C01813=1150.648,329.921,-76.910,-176.647,8.812,148.784
C01814=1150.652,329.674,-76.877,-176.650,8.808,148.783
C01815=1150.656,329.426,-76.845,-176.652,8.805,148.783
C01816=1150.660,329.178,-76.812,-176.654,8.801,148.783
C01817=1150.664,328.930,-76.779,-176.657,8.797,148.783
C01818=1150.668,328.682,-76.746,-176.659,8.794,148.783
C01819=1150.672,328.434,-76.713,-176.662,8.790,148.782
C01820=1150.676,328.187,-76.681,-176.665,8.787,148.782
C01821=1150.680,327.939,-76.648,-176.667,8.783,148.782
C01822=1150.684,327.690,-76.615,-176.670,8.779,148.782
C01823=1150.688,327.443,-76.582,-176.672,8.776,148.782
C01824=1150.692,327.195,-76.549,-176.675,8.772,148.781
C01825=1150.696,326.947,-76.517,-176.677,8.769,148.781
C01826=1150.700,326.699,-76.484,-176.680,8.765,148.781
C01827=1150.704,326.451,-76.452,-176.683,8.761,148.781
C01828=1150.708,326.203,-76.419,-176.685,8.758,148.781
C01829=1150.712,325.956,-76.386,-176.687,8.755,148.780
C01830=1150.717,325.708,-76.354,-176.690,8.751,148.780
C01831=1150.721,325.461,-76.321,-176.693,8.748,148.780
C01832=1150.725,325.212,-76.289,-176.696,8.744,148.780
C01833=1150.729,324.965,-76.256,-176.698,8.740,148.780
C01834=1150.733,324.717,-76.224,-176.700,8.737,148.780
C01835=1150.737,324.469,-76.190,-176.703,8.733,148.779
C01836=1150.741,324.221,-76.159,-176.706,8.730,148.779
C01837=1150.745,323.973,-76.125,-176.708,8.727,148.779
C01838=1150.749,323.726,-76.094,-176.711,8.722,148.779
C01839=1150.754,323.477,-76.062,-176.713,8.719,148.778
C01840=1150.758,323.230,-76.028,-176.716,8.715,148.778
C01841=1150.762,322.982,-75.997,-176.718,8.712,148.778
C01842=1150.766,322.734,-75.963,-176.721,8.709,148.778
C01843=1150.770,322.486,-75.932,-176.724,8.704,148.778
C01844=1150.774,322.237,-75.899,-176.726,8.701,148.778
C01845=1150.778,321.991,-75.867,-176.729,8.698,148.777
C01846=1150.783,321.742,-75.834,-176.732,8.694,148.777
C01847=1150.786,321.494,-75.803,-176.734,8.691,148.777
C01848=1150.790,321.247,-75.769,-176.736,8.688,148.777
C01849=1150.794,320.999,-75.738,-176.739,8.683,148.777
C01850=1150.799,320.751,-75.706,-176.742,8.680,148.776
C01851=1150.803,320.503,-75.674,-176.744,8.677,148.776
C01852=1150.807,320.255,-75.641,-176.747,8.673,148.776
C01853=1150.811,320.007,-75.609,-176.750,8.670,148.776
C01854=1150.815,319.759,-75.576,-176.752,8.667,148.776
C01855=1150.819,319.511,-75.545,-176.755,8.663,148.776
C01856=1150.823,319.263,-75.513,-176.757,8.659,148.775
C01857=1150.827,319.016,-75.480,-176.759,8.656,148.775
C01858=1150.831,318.768,-75.448,-176.762,8.652,148.775
C01859=1150.836,318.520,-75.416,-176.765,8.649,148.775
C01860=1150.840,318.272,-75.384,-176.767,8.646,148.775
C01861=1150.843,318.024,-75.352,-176.770,8.642,148.775
C01862=1150.848,317.776,-75.320,-176.773,8.638,148.774
C01863=1150.852,317.528,-75.288,-176.775,8.635,148.774
C01864=1150.857,317.280,-75.256,-176.778,8.631,148.774
C01865=1150.860,317.032,-75.224,-176.781,8.628,148.774
C01866=1150.865,316.785,-75.192,-176.783,8.625,148.774
C01867=1150.869,316.536,-75.160,-176.786,8.621,148.774
C01868=1150.873,316.288,-75.128,-176.788,8.617,148.773
C01869=1150.877,316.041,-75.097,-176.790,8.614,148.773
C01870=1150.881,315.793,-75.065,-176.794,8.610,148.773
C01871=1150.885,315.544,-75.032,-176.796,8.607,148.773
C01872=1150.890,315.297,-75.001,-176.798,8.604,148.773
C01873=1150.893,315.049,-74.969,-176.801,8.600,148.773
C01874=1150.898,314.801,-74.937,-176.804,8.596,148.772
C01875=1150.902,314.553,-74.905,-176.806,8.593,148.772
C01876=1150.906,314.305,-74.873,-176.809,8.590,148.772
C01877=1150.909,314.057,-74.841,-176.812,8.586,148.772
C01878=1150.914,313.779,-74.805,-176.814,8.583,148.772
C01879=1150.919,313.503,-74.770,-176.817,8.579,148.772
C01880=1150.924,313.224,-74.735,-176.820,8.575,148.772
C01881=1150.928,312.947,-74.700,-176.823,8.571,148.771
C01882=1150.932,312.699,-74.668,-176.825,8.568,148.771
C01883=1150.936,312.452,-74.636,-176.828,8.564,148.771
C01884=1150.941,312.203,-74.604,-176.831,8.561,148.771
C01885=1150.945,311.955,-74.573,-176.833,8.557,148.771
C01886=1150.949,311.707,-74.541,-176.836,8.554,148.771
C01887=1150.953,311.460,-74.510,-176.839,8.550,148.771
C01888=1150.957,311.212,-74.478,-176.841,8.547,148.770
C01889=1150.961,310.963,-74.447,-176.844,8.544,148.770
C01890=1150.966,310.716,-74.415,-176.846,8.540,148.770
C01891=1150.970,310.467,-74.383,-176.849,8.537,148.770
C01892=1150.974,310.220,-74.352,-176.852,8.533,148.770
C01893=1150.978,309.971,-74.320,-176.854,8.530,148.770
C01894=1150.983,309.724,-74.289,-176.857,8.526,148.769
C01895=1150.987,309.475,-74.258,-176.860,8.523,148.769
C01896=1150.991,309.228,-74.226,-176.862,8.520,148.769
C01897=1150.995,308.980,-74.195,-176.864,8.516,148.769
C01898=1150.999,308.731,-74.163,-176.868,8.513,148.769
C01899=1151.003,308.484,-74.132,-176.870,8.509,148.769
C01900=1151.007,308.235,-74.100,-176.872,8.506,148.769
C01901=1151.011,307.988,-74.069,-176.875,8.503,148.768
C01902=1151.015,307.739,-74.038,-176.878,8.499,148.768
C01903=1151.020,307.492,-74.006,-176.880,8.496,148.768
C01904=1151.024,307.243,-73.975,-176.883,8.493,148.768
C01905=1151.029,306.996,-73.943,-176.885,8.490,148.768
C01906=1151.033,306.747,-73.912,-176.888,8.486,148.768
C01907=1151.037,306.500,-73.881,-176.891,8.482,148.768
C01908=1151.041,306.252,-73.850,-176.893,8.479,148.768
C01909=1151.045,306.004,-73.819,-176.896,8.476,148.768
C01910=1151.049,305.756,-73.788,-176.899,8.472,148.767
C01911=1151.053,305.508,-73.757,-176.901,8.469,148.767
C01912=1151.057,305.260,-73.725,-176.904,8.466,148.767
C01913=1151.061,305.012,-73.694,-176.906,8.462,148.767
C01914=1151.066,304.764,-73.663,-176.909,8.459,148.767
C01915=1151.070,304.516,-73.631,-176.912,8.455,148.767
C01916=1151.074,304.268,-73.601,-176.914,8.452,148.767
C01917=1151.079,304.020,-73.570,-176.917,8.449,148.767
C01918=1151.083,303.772,-73.538,-176.920,8.445,148.766
C01919=1151.087,303.524,-73.507,-176.922,8.442,148.766
C01920=1151.091,303.275,-73.476,-176.925,8.439,148.766
C01921=1151.095,303.027,-73.446,-176.927,8.436,148.766
C01922=1151.099,302.780,-73.415,-176.930,8.432,148.766
C01923=1151.103,302.531,-73.383,-176.933,8.429,148.766
C01924=1151.108,302.283,-73.353,-176.935,8.426,148.766
C01925=1151.112,302.035,-73.322,-176.938,8.422,148.766
C01926=1151.117,301.787,-73.291,-176.940,8.419,148.766
C01927=1151.121,301.539,-73.261,-176.943,8.415,148.766
C01928=1151.124,301.291,-73.229,-176.946,8.412,148.765
C01929=1151.129,301.043,-73.198,-176.949,8.409,148.765
C01930=1151.134,300.795,-73.167,-176.951,8.406,148.765
C01931=1151.138,300.546,-73.136,-176.954,8.402,148.765
C01932=1151.141,300.299,-73.106,-176.957,8.399,148.765
C01933=1151.146,300.051,-73.075,-176.959,8.396,148.765
C01934=1151.150,299.802,-73.044,-176.962,8.393,148.765
C01935=1151.155,299.554,-73.013,-176.964,8.389,148.765
C01936=1151.159,299.307,-72.983,-176.967,8.385,148.765
C01937=1151.163,299.058,-72.952,-176.970,8.382,148.765
C01938=1151.167,298.810,-72.921,-176.972,8.379,148.764
C01939=1151.171,298.562,-72.891,-176.975,8.376,148.764
C01940=1151.175,298.314,-72.860,-176.977,8.373,148.764
C01941=1151.180,298.066,-72.829,-176.980,8.369,148.764
C01942=1151.184,297.818,-72.799,-176.983,8.366,148.764
C01943=1151.188,297.570,-72.768,-176.985,8.363,148.764
C01944=1151.192,297.321,-72.737,-176.988,8.360,148.764
C01945=1151.196,297.074,-72.707,-176.990,8.356,148.764
C01946=1151.201,296.826,-72.676,-176.993,8.352,148.764
C01947=1151.205,296.578,-72.645,-176.996,8.349,148.764
C01948=1151.209,296.330,-72.615,-176.999,8.346,148.764
C01949=1151.213,296.082,-72.584,-177.001,8.343,148.763
C01950=1151.217,295.834,-72.554,-177.004,8.340,148.763
C01951=1151.222,295.585,-72.524,-177.006,8.337,148.763
C01952=1151.225,295.337,-72.493,-177.009,8.333,148.763
C01953=1151.230,295.089,-72.463,-177.012,8.330,148.763
C01954=1151.234,294.841,-72.432,-177.014,8.327,148.763
C01955=1151.238,294.593,-72.402,-177.017,8.324,148.763
C01956=1151.243,294.344,-72.371,-177.019,8.321,148.763
C01957=1151.246,294.097,-72.341,-177.022,8.316,148.763
C01958=1151.251,293.849,-72.310,-177.025,8.314,148.763
C01959=1151.255,293.601,-72.280,-177.027,8.310,148.763
C01960=1151.260,293.352,-72.250,-177.030,8.307,148.763
C01961=1151.263,293.104,-72.220,-177.033,8.304,148.762
C01962=1151.268,292.856,-72.189,-177.035,8.301,148.763
C01963=1151.272,292.608,-72.159,-177.038,8.297,148.762
C01964=1151.277,292.360,-72.129,-177.041,8.294,148.762
C01965=1151.280,292.112,-72.098,-177.043,8.291,148.762
C01966=1151.285,291.863,-72.068,-177.046,8.288,148.762
C01967=1151.289,291.615,-72.038,-177.048,8.285,148.762
C01968=1151.293,291.367,-72.008,-177.051,8.282,148.762
C01969=1151.297,291.119,-71.978,-177.054,8.278,148.762
C01970=1151.301,290.871,-71.947,-177.057,8.275,148.762
C01971=1151.306,290.623,-71.917,-177.060,8.272,148.762
C01972=1151.310,290.375,-71.887,-177.062,8.268,148.762
C01973=1151.314,290.126,-71.857,-177.065,8.265,148.762
C01974=1151.318,289.878,-71.827,-177.067,8.262,148.762
C01975=1151.322,289.630,-71.797,-177.070,8.259,148.762
C01976=1151.327,289.382,-71.766,-177.073,8.255,148.761
C01977=1151.331,289.134,-71.737,-177.075,8.252,148.762
C01978=1151.335,288.886,-71.707,-177.078,8.249,148.762
C01979=1151.340,288.637,-71.677,-177.081,8.246,148.761
C01980=1151.344,288.390,-71.647,-177.083,8.243,148.761
C01981=1151.348,288.142,-71.617,-177.086,8.240,148.761
C01982=1151.352,287.866,-71.583,-177.089,8.236,148.761
C01983=1151.358,287.590,-71.550,-177.092,8.233,148.761
C01984=1151.363,287.316,-71.517,-177.095,8.229,148.761
C01985=1151.367,287.040,-71.484,-177.098,8.225,148.761
C01986=1151.371,286.793,-71.454,-177.101,8.222,148.761
C01987=1151.376,286.544,-71.425,-177.103,8.219,148.761
C01988=1151.380,286.296,-71.395,-177.106,8.216,148.761
C01989=1151.384,286.047,-71.364,-177.108,8.213,148.761
C01990=1151.388,285.799,-71.335,-177.111,8.210,148.761
C01991=1151.392,285.551,-71.305,-177.114,8.207,148.761
C01992=1151.397,285.302,-71.275,-177.117,8.203,148.761
C01993=1151.401,285.055,-71.245,-177.119,8.200,148.761
C01994=1151.405,284.806,-71.216,-177.122,8.197,148.761
C01995=1151.409,284.558,-71.186,-177.124,8.194,148.761
C01996=1151.413,284.310,-71.157,-177.127,8.191,148.761
C01997=1151.418,284.062,-71.127,-177.130,8.187,148.761
C01998=1151.422,283.814,-71.096,-177.132,8.184,148.761
C01999=1151.426,283.565,-71.067,-177.135,8.181,148.761
C02000=1151.431,283.318,-71.038,-177.137,8.178,148.760
C02001=1151.435,283.070,-71.008,-177.141,8.174,148.760
C02002=1151.440,282.821,-70.979,-177.144,8.172,148.760
C02003=1151.444,282.573,-70.950,-177.146,8.168,148.760
C02004=1151.449,282.324,-70.919,-177.149,8.165,148.760
C02005=1151.453,282.076,-70.890,-177.151,8.162,148.760
C02006=1151.457,281.829,-70.860,-177.154,8.159,148.760
C02007=1151.461,281.580,-70.830,-177.156,8.156,148.760
C02008=1151.465,281.332,-70.801,-177.159,8.153,148.760
C02009=1151.469,281.084,-70.771,-177.162,8.150,148.760
C02010=1151.473,280.835,-70.742,-177.164,8.147,148.760
C02011=1151.478,280.587,-70.713,-177.168,8.143,148.760
C02012=1151.482,280.339,-70.683,-177.170,8.140,148.760
C02013=1151.486,280.091,-70.654,-177.173,8.137,148.760
C02014=1151.491,279.843,-70.625,-177.176,8.134,148.760
C02015=1151.495,279.594,-70.596,-177.178,8.131,148.760
C02016=1151.499,279.346,-70.566,-177.181,8.128,148.760
C02017=1151.504,279.098,-70.537,-177.183,8.125,148.760
C02018=1151.508,278.849,-70.507,-177.186,8.122,148.760
C02019=1151.512,278.601,-70.478,-177.188,8.119,148.760
C02020=1151.516,278.353,-70.449,-177.191,8.116,148.760
C02021=1151.520,278.105,-70.419,-177.194,8.112,148.760
C02022=1151.524,277.856,-70.390,-177.196,8.110,148.760
C02023=1151.529,277.609,-70.361,-177.200,8.106,148.760
C02024=1151.534,277.360,-70.332,-177.202,8.103,148.760
C02025=1151.538,277.112,-70.302,-177.205,8.100,148.760
C02026=1151.542,276.863,-70.273,-177.208,8.097,148.760
C02027=1151.546,276.615,-70.243,-177.210,8.094,148.760
C02028=1151.550,276.367,-70.214,-177.213,8.091,148.760
C02029=1151.555,276.119,-70.186,-177.215,8.087,148.760
C02030=1151.559,275.871,-70.157,-177.218,8.085,148.760
C02031=1151.563,275.622,-70.127,-177.221,8.082,148.760
C02032=1151.568,275.373,-70.099,-177.223,8.078,148.760
C02033=1151.572,275.125,-70.069,-177.226,8.075,148.760
C02034=1151.577,274.878,-70.040,-177.229,8.072,148.760
C02035=1151.581,274.629,-70.011,-177.232,8.069,148.760
C02036=1151.585,274.381,-69.982,-177.234,8.066,148.760
C02037=1151.589,274.133,-69.953,-177.237,8.063,148.760
C02038=1151.593,273.884,-69.924,-177.239,8.060,148.760
C02039=1151.598,273.636,-69.895,-177.243,8.057,148.760
C02040=1151.602,273.388,-69.866,-177.246,8.054,148.760
C02041=1151.606,273.139,-69.838,-177.248,8.050,148.760
C02042=1151.610,272.891,-69.808,-177.251,8.047,148.760
C02043=1151.615,272.643,-69.780,-177.253,8.044,148.760
C02044=1151.619,272.395,-69.750,-177.256,8.042,148.760
C02045=1151.623,272.146,-69.722,-177.259,8.038,148.760
C02046=1151.628,271.898,-69.693,-177.261,8.035,148.760
C02047=1151.632,271.649,-69.664,-177.264,8.032,148.760
C02048=1151.637,271.401,-69.635,-177.267,8.029,148.760
C02049=1151.640,271.153,-69.607,-177.270,8.026,148.760
C02050=1151.645,270.905,-69.578,-177.272,8.023,148.760
C02051=1151.650,270.656,-69.549,-177.275,8.020,148.760
C02052=1151.653,270.408,-69.520,-177.278,8.017,148.760
C02053=1151.658,270.160,-69.492,-177.280,8.014,148.760
C02054=1151.662,269.912,-69.462,-177.283,8.011,148.760
C02055=1151.666,269.663,-69.434,-177.285,8.008,148.760
C02056=1151.671,269.415,-69.406,-177.288,8.005,148.760
C02057=1151.675,269.167,-69.376,-177.291,8.002,148.760
C02058=1151.679,268.918,-69.348,-177.294,7.999,148.760
C02059=1151.684,268.670,-69.320,-177.296,7.996,148.760
C02060=1151.688,268.422,-69.290,-177.299,7.993,148.760
C02061=1151.692,268.173,-69.262,-177.302,7.990,148.760
C02062=1151.697,267.925,-69.234,-177.304,7.987,148.760
C02063=1151.701,267.677,-69.204,-177.307,7.984,148.760
C02064=1151.705,267.428,-69.176,-177.310,7.981,148.760
C02065=1151.710,267.180,-69.148,-177.313,7.978,148.760
C02066=1151.714,266.931,-69.120,-177.315,7.976,148.760
C02067=1151.719,266.684,-69.091,-177.318,7.972,148.760
C02068=1151.723,266.435,-69.062,-177.321,7.969,148.760
C02069=1151.727,266.186,-69.034,-177.323,7.966,148.760
C02070=1151.731,265.938,-69.006,-177.326,7.963,148.760
C02071=1151.736,265.690,-68.977,-177.329,7.960,148.760
C02072=1151.741,265.442,-68.948,-177.332,7.958,148.760
C02073=1151.744,265.193,-68.920,-177.334,7.955,148.760
C02074=1151.749,264.945,-68.891,-177.337,7.951,148.760
C02075=1151.753,264.697,-68.863,-177.339,7.948,148.760
C02076=1151.758,264.448,-68.835,-177.342,7.945,148.760
C02077=1151.762,264.200,-68.807,-177.345,7.943,148.760
C02078=1151.766,263.951,-68.779,-177.348,7.940,148.760
C02079=1151.771,263.703,-68.750,-177.351,7.937,148.761
C02080=1151.775,263.455,-68.722,-177.353,7.934,148.761
C02081=1151.780,263.206,-68.694,-177.356,7.931,148.761
C02082=1151.783,262.958,-68.665,-177.358,7.927,148.761
C02083=1151.788,262.710,-68.637,-177.361,7.925,148.761
C02084=1151.792,262.462,-68.609,-177.364,7.922,148.761
C02085=1151.797,262.213,-68.580,-177.367,7.919,148.761
C02086=1151.802,261.940,-68.549,-177.370,7.915,148.761
C02087=1151.806,261.666,-68.518,-177.373,7.912,148.761
C02088=1151.811,261.393,-68.488,-177.376,7.909,148.761
C02089=1151.816,261.119,-68.456,-177.379,7.905,148.761
C02090=1151.820,260.871,-68.429,-177.382,7.902,148.761
C02091=1151.824,260.623,-68.401,-177.385,7.899,148.761
C02092=1151.829,260.374,-68.372,-177.387,7.896,148.761
C02093=1151.833,260.126,-68.344,-177.390,7.894,148.761
C02094=1151.837,259.878,-68.316,-177.393,7.891,148.761
C02095=1151.842,259.629,-68.288,-177.396,7.888,148.761
C02096=1151.846,259.381,-68.260,-177.398,7.886,148.761
C02097=1151.851,259.133,-68.233,-177.400,7.882,148.761
C02098=1151.854,258.884,-68.205,-177.403,7.879,148.761
C02099=1151.860,258.636,-68.176,-177.406,7.876,148.761
C02100=1151.863,258.387,-68.148,-177.409,7.873,148.761
C02101=1151.868,258.139,-68.121,-177.411,7.871,148.761
C02102=1151.872,257.890,-68.093,-177.414,7.868,148.761
C02103=1151.877,257.642,-68.064,-177.417,7.865,148.762
C02104=1151.881,257.394,-68.037,-177.420,7.862,148.762
C02105=1151.885,257.145,-68.009,-177.422,7.859,148.762
C02106=1151.890,256.897,-67.981,-177.425,7.856,148.762
C02107=1151.894,256.648,-67.953,-177.428,7.853,148.762
C02108=1151.899,256.400,-67.926,-177.431,7.850,148.762
C02109=1151.903,256.152,-67.898,-177.434,7.847,148.762
C02110=1151.907,255.903,-67.870,-177.436,7.844,148.762
C02111=1151.911,255.655,-67.843,-177.439,7.841,148.762
C02112=1151.916,255.407,-67.815,-177.442,7.838,148.762
C02113=1151.921,255.157,-67.787,-177.445,7.835,148.762
C02114=1151.925,254.910,-67.759,-177.447,7.832,148.762
C02115=1151.929,254.661,-67.731,-177.450,7.830,148.762
C02116=1151.933,254.413,-67.704,-177.452,7.827,148.762
C02117=1151.938,254.165,-67.676,-177.455,7.824,148.762
C02118=1151.942,253.915,-67.649,-177.458,7.821,148.763
C02119=1151.946,253.668,-67.621,-177.461,7.818,148.763
C02120=1151.951,253.419,-67.594,-177.464,7.816,148.763
C02121=1151.955,253.170,-67.565,-177.466,7.813,148.763
C02122=1151.960,252.922,-67.538,-177.469,7.810,148.763
C02123=1151.964,252.674,-67.510,-177.472,7.807,148.763
C02124=1151.969,252.425,-67.483,-177.475,7.804,148.763
C02125=1151.973,252.177,-67.455,-177.477,7.801,148.763
C02126=1151.977,251.928,-67.428,-177.480,7.798,148.763
C02127=1151.982,251.680,-67.400,-177.483,7.795,148.763
C02128=1151.986,251.431,-67.373,-177.485,7.793,148.763
C02129=1151.990,251.183,-67.346,-177.488,7.790,148.763
C02130=1151.995,250.935,-67.318,-177.491,7.787,148.763
C02131=1151.999,250.686,-67.291,-177.494,7.784,148.763
C02132=1152.003,250.437,-67.263,-177.496,7.781,148.764
C02133=1152.008,250.189,-67.236,-177.499,7.778,148.764
C02134=1152.012,249.941,-67.209,-177.502,7.775,148.764
C02135=1152.017,249.692,-67.182,-177.505,7.772,148.764
C02136=1152.021,249.444,-67.153,-177.507,7.769,148.764
C02137=1152.026,249.195,-67.126,-177.510,7.766,148.764
C02138=1152.030,248.947,-67.099,-177.512,7.764,148.764
C02139=1152.035,248.699,-67.072,-177.515,7.761,148.764
C02140=1152.038,248.450,-67.045,-177.518,7.758,148.764
C02141=1152.042,248.201,-67.018,-177.521,7.756,148.764
C02142=1152.047,247.953,-66.991,-177.524,7.753,148.764
C02143=1152.052,247.704,-66.964,-177.526,7.750,148.764
C02144=1152.056,247.457,-66.936,-177.529,7.747,148.764
C02145=1152.060,247.207,-66.908,-177.532,7.744,148.764
C02146=1152.065,246.959,-66.881,-177.535,7.741,148.765
C02147=1152.070,246.710,-66.854,-177.537,7.739,148.765
C02148=1152.074,246.462,-66.827,-177.540,7.736,148.765
C02149=1152.078,246.214,-66.801,-177.543,7.733,148.765
C02150=1152.083,245.965,-66.774,-177.546,7.730,148.765
C02151=1152.087,245.717,-66.745,-177.548,7.727,148.765
C02152=1152.091,245.468,-66.718,-177.551,7.724,148.765
C02153=1152.096,245.220,-66.691,-177.554,7.721,148.765
C02154=1152.100,244.971,-66.665,-177.557,7.719,148.765
C02155=1152.104,244.723,-66.638,-177.559,7.716,148.765
C02156=1152.109,244.474,-66.611,-177.562,7.714,148.766
C02157=1152.113,244.225,-66.583,-177.565,7.711,148.766
C02158=1152.118,243.977,-66.556,-177.567,7.708,148.766
C02159=1152.122,243.729,-66.530,-177.570,7.705,148.766
C02160=1152.126,243.480,-66.503,-177.573,7.702,148.766
C02161=1152.131,243.232,-66.476,-177.576,7.699,148.766
C02162=1152.136,242.983,-66.449,-177.578,7.697,148.766
C02163=1152.140,242.735,-66.422,-177.581,7.694,148.766
C02164=1152.144,242.486,-66.395,-177.584,7.691,148.766
C02165=1152.149,242.238,-66.368,-177.587,7.688,148.766
C02166=1152.153,241.989,-66.342,-177.589,7.685,148.767
C02167=1152.157,241.740,-66.315,-177.592,7.682,148.767
C02168=1152.162,241.491,-66.288,-177.594,7.680,148.767
C02169=1152.166,241.243,-66.261,-177.598,7.678,148.767
C02170=1152.170,240.995,-66.234,-177.600,7.675,148.767
C02171=1152.175,240.746,-66.207,-177.603,7.672,148.767
C02172=1152.179,240.498,-66.181,-177.606,7.669,148.767
C02173=1152.184,240.249,-66.154,-177.609,7.666,148.767
C02174=1152.189,240.000,-66.127,-177.612,7.663,148.767
C02175=1152.193,239.752,-66.101,-177.614,7.661,148.767
C02176=1152.197,239.504,-66.074,-177.617,7.658,148.768
C02177=1152.201,239.256,-66.047,-177.620,7.655,148.768
C02178=1152.206,239.006,-66.021,-177.623,7.652,148.768
C02179=1152.211,238.758,-65.994,-177.625,7.650,148.768
C02180=1152.215,238.510,-65.967,-177.628,7.647,148.768
C02181=1152.220,238.261,-65.941,-177.630,7.644,148.768
C02182=1152.224,238.013,-65.915,-177.633,7.642,148.768
C02183=1152.228,237.764,-65.888,-177.636,7.639,148.769
C02184=1152.232,237.515,-65.862,-177.639,7.636,148.769
C02185=1152.237,237.267,-65.835,-177.642,7.633,148.769
C02186=1152.241,237.019,-65.808,-177.644,7.631,148.769
C02187=1152.246,236.769,-65.782,-177.647,7.628,148.769
C02188=1152.250,236.521,-65.756,-177.650,7.625,148.769
C02189=1152.255,236.273,-65.728,-177.653,7.623,148.769
C02190=1152.260,236.001,-65.700,-177.656,7.620,148.769
C02191=1152.264,235.729,-65.671,-177.659,7.617,148.769
C02192=1152.270,235.457,-65.642,-177.661,7.614,148.770
C02193=1152.274,235.186,-65.614,-177.665,7.611,148.770
C02194=1152.279,234.937,-65.587,-177.667,7.608,148.770
C02195=1152.283,234.688,-65.561,-177.670,7.605,148.770
C02196=1152.288,234.440,-65.534,-177.673,7.602,148.770
C02197=1152.292,234.191,-65.508,-177.676,7.599,148.770
C02198=1152.296,233.943,-65.482,-177.678,7.598,148.770
C02199=1152.301,233.694,-65.455,-177.681,7.595,148.771
C02200=1152.305,233.445,-65.429,-177.684,7.592,148.771
C02201=1152.310,233.197,-65.402,-177.687,7.589,148.771
C02202=1152.314,232.948,-65.377,-177.689,7.586,148.771
C02203=1152.318,232.700,-65.351,-177.692,7.584,148.771
C02204=1152.323,232.451,-65.324,-177.695,7.581,148.771
C02205=1152.327,232.203,-65.298,-177.698,7.578,148.771
C02206=1152.332,231.954,-65.272,-177.701,7.575,148.771
C02207=1152.336,231.705,-65.246,-177.703,7.573,148.771
C02208=1152.340,231.457,-65.219,-177.706,7.571,148.772
C02209=1152.345,231.209,-65.194,-177.709,7.568,148.772
C02210=1152.350,230.960,-65.167,-177.712,7.565,148.772
C02211=1152.354,230.711,-65.141,-177.714,7.562,148.772
C02212=1152.358,230.463,-65.115,-177.717,7.560,148.772
C02213=1152.363,230.214,-65.089,-177.720,7.557,148.772
C02214=1152.368,229.965,-65.063,-177.723,7.554,148.773
C02215=1152.372,229.717,-65.037,-177.725,7.551,148.773
C02216=1152.376,229.468,-65.011,-177.728,7.549,148.773
C02217=1152.381,229.219,-64.985,-177.731,7.547,148.773
C02218=1152.385,228.971,-64.959,-177.734,7.544,148.773
C02219=1152.389,228.722,-64.933,-177.736,7.541,148.773
C02220=1152.394,228.474,-64.907,-177.739,7.539,148.773
C02221=1152.399,228.225,-64.881,-177.742,7.536,148.774
C02222=1152.403,227.976,-64.855,-177.745,7.533,148.774
C02223=1152.408,227.727,-64.829,-177.747,7.530,148.774
C02224=1152.412,227.479,-64.804,-177.750,7.528,148.774
C02225=1152.417,227.231,-64.778,-177.753,7.526,148.774
C02226=1152.421,226.982,-64.751,-177.756,7.523,148.774
C02227=1152.426,226.733,-64.726,-177.758,7.520,148.774
C02228=1152.430,226.484,-64.700,-177.761,7.518,148.774
C02229=1152.435,226.236,-64.674,-177.764,7.515,148.775
C02230=1152.439,225.988,-64.649,-177.767,7.512,148.775
C02231=1152.443,225.739,-64.623,-177.769,7.510,148.775
C02232=1152.447,225.490,-64.597,-177.772,7.507,148.775
C02233=1152.453,225.242,-64.571,-177.775,7.504,148.775
C02234=1152.457,224.993,-64.545,-177.778,7.502,148.775
C02235=1152.461,224.744,-64.520,-177.780,7.499,148.776
C02236=1152.466,224.496,-64.494,-177.783,7.497,148.776
C02237=1152.470,224.247,-64.469,-177.786,7.494,148.776
C02238=1152.475,223.998,-64.443,-177.789,7.491,148.776
C02239=1152.479,223.750,-64.417,-177.791,7.489,148.776
C02240=1152.484,223.501,-64.392,-177.794,7.486,148.776
C02241=1152.488,223.253,-64.366,-177.797,7.483,148.777
C02242=1152.492,223.004,-64.340,-177.799,7.481,148.777
C02243=1152.497,222.755,-64.315,-177.802,7.479,148.777
C02244=1152.501,222.506,-64.290,-177.805,7.476,148.777
C02245=1152.506,222.258,-64.264,-177.807,7.474,148.777
C02246=1152.510,222.009,-64.239,-177.811,7.471,148.778
C02247=1152.515,221.760,-64.213,-177.813,7.468,148.778
C02248=1152.520,221.512,-64.187,-177.816,7.465,148.778
C02249=1152.524,221.264,-64.162,-177.818,7.463,148.778
C02250=1152.528,221.014,-64.137,-177.822,7.460,148.778
C02251=1152.533,220.766,-64.111,-177.824,7.458,148.778
C02252=1152.537,220.517,-64.086,-177.827,7.455,148.778
C02253=1152.542,220.268,-64.060,-177.830,7.453,148.779
C02254=1152.547,220.020,-64.035,-177.833,7.450,148.779
C02255=1152.551,219.771,-64.009,-177.835,7.448,148.779
C02256=1152.556,219.523,-63.984,-177.838,7.445,148.779
C02257=1152.560,219.274,-63.958,-177.841,7.442,148.779
C02258=1152.564,219.025,-63.933,-177.843,7.440,148.779
C02259=1152.569,218.776,-63.908,-177.846,7.438,148.780
C02260=1152.574,218.528,-63.882,-177.849,7.435,148.780
C02261=1152.578,218.279,-63.858,-177.851,7.433,148.780
C02262=1152.582,218.030,-63.832,-177.855,7.430,148.780
C02263=1152.587,217.782,-63.807,-177.857,7.427,148.780
C02264=1152.592,217.533,-63.782,-177.860,7.425,148.780
C02265=1152.596,217.284,-63.756,-177.863,7.422,148.781
C02266=1152.601,217.035,-63.731,-177.866,7.420,148.781
C02267=1152.604,216.787,-63.706,-177.868,7.417,148.781
C02268=1152.609,216.539,-63.681,-177.871,7.415,148.781
C02269=1152.614,216.289,-63.656,-177.874,7.412,148.781
C02270=1152.619,216.041,-63.630,-177.877,7.410,148.782
C02271=1152.623,215.792,-63.605,-177.879,7.407,148.782
C02272=1152.627,215.544,-63.581,-177.882,7.404,148.782
C02273=1152.632,215.295,-63.556,-177.885,7.403,148.782
C02274=1152.637,215.047,-63.530,-177.888,7.400,148.782
C02275=1152.641,214.797,-63.505,-177.890,7.397,148.782
C02276=1152.646,214.549,-63.480,-177.893,7.395,148.783
C02277=1152.650,214.300,-63.455,-177.896,7.392,148.783
C02278=1152.654,214.052,-63.430,-177.899,7.390,148.783
C02279=1152.659,213.802,-63.405,-177.901,7.387,148.783
C02280=1152.663,213.555,-63.380,-177.904,7.384,148.783
C02281=1152.668,213.305,-63.355,-177.907,7.383,148.784
C02282=1152.673,213.056,-63.330,-177.910,7.380,148.784
C02283=1152.677,212.808,-63.305,-177.912,7.377,148.784
C02284=1152.681,212.559,-63.281,-177.915,7.375,148.784
C02285=1152.686,212.310,-63.256,-177.918,7.372,148.784
C02286=1152.691,212.062,-63.230,-177.921,7.370,148.785
C02287=1152.695,211.813,-63.206,-177.923,7.367,148.785
C02288=1152.700,211.564,-63.181,-177.926,7.364,148.785
C02289=1152.704,211.316,-63.156,-177.929,7.363,148.785
C02290=1152.708,211.067,-63.131,-177.932,7.360,148.785
C02291=1152.713,210.818,-63.107,-177.935,7.357,148.786
C02292=1152.717,210.569,-63.081,-177.937,7.355,148.786
C02293=1152.722,210.321,-63.057,-177.940,7.352,148.786
C02294=1152.727,210.050,-63.030,-177.943,7.350,148.786
C02295=1152.732,209.780,-63.003,-177.946,7.347,148.786
C02296=1152.737,209.509,-62.976,-177.949,7.345,148.787
C02297=1152.741,209.239,-62.949,-177.952,7.342,148.787
C02298=1152.747,208.990,-62.924,-177.955,7.339,148.787
C02299=1152.750,208.741,-62.900,-177.957,7.337,148.787
C02300=1152.755,208.492,-62.875,-177.960,7.335,148.787
C02301=1152.761,208.243,-62.851,-177.963,7.332,148.788
C02302=1152.764,207.994,-62.826,-177.966,7.330,148.788
C02303=1152.769,207.746,-62.801,-177.968,7.327,148.788
C02304=1152.774,207.498,-62.777,-177.972,7.325,148.788
C02305=1152.778,207.248,-62.752,-177.974,7.322,148.788
C02306=1152.783,207.000,-62.728,-177.977,7.320,148.789
C02307=1152.788,206.751,-62.703,-177.979,7.318,148.789
C02308=1152.791,206.502,-62.679,-177.982,7.315,148.789
C02309=1152.797,206.253,-62.654,-177.985,7.313,148.789
C02310=1152.801,206.005,-62.630,-177.988,7.310,148.789
C02311=1152.806,205.755,-62.605,-177.991,7.308,148.790
C02312=1152.810,205.507,-62.581,-177.993,7.306,148.790
C02313=1152.815,205.258,-62.556,-177.996,7.303,148.790
C02314=1152.819,205.009,-62.532,-177.999,7.301,148.790
C02315=1152.823,204.761,-62.508,-178.002,7.298,148.791
C02316=1152.828,204.512,-62.483,-178.004,7.296,148.791
C02317=1152.833,204.264,-62.459,-178.007,7.294,148.791
C02318=1152.837,204.014,-62.434,-178.010,7.291,148.791
C02319=1152.842,203.766,-62.410,-178.013,7.289,148.792
C02320=1152.846,203.517,-62.386,-178.016,7.286,148.792
C02321=1152.851,203.269,-62.361,-178.018,7.284,148.792
C02322=1152.855,203.020,-62.337,-178.021,7.281,148.792
C02323=1152.860,202.770,-62.313,-178.024,7.280,148.792
C02324=1152.865,202.522,-62.288,-178.027,7.277,148.793
C02325=1152.869,202.273,-62.264,-178.029,7.275,148.793
C02326=1152.874,202.024,-62.239,-178.032,7.272,148.793
C02327=1152.878,201.776,-62.215,-178.034,7.270,148.793
C02328=1152.883,201.527,-62.191,-178.037,7.267,148.794
C02329=1152.887,201.278,-62.168,-178.040,7.265,148.794
C02330=1152.892,201.029,-62.143,-178.043,7.263,148.794
C02331=1152.896,200.780,-62.119,-178.046,7.260,148.794
C02332=1152.901,200.532,-62.095,-178.048,7.258,148.794
C02333=1152.906,200.283,-62.070,-178.051,7.255,148.795
C02334=1152.910,200.034,-62.047,-178.054,7.253,148.795
C02335=1152.914,199.785,-62.022,-178.057,7.251,148.795
C02336=1152.919,199.537,-61.998,-178.059,7.249,148.795
C02337=1152.924,199.287,-61.974,-178.063,7.246,148.796
C02338=1152.928,199.039,-61.950,-178.065,7.244,148.796
C02339=1152.933,198.790,-61.926,-178.068,7.241,148.796
C02340=1152.938,198.541,-61.903,-178.070,7.239,148.796
C02341=1152.942,198.292,-61.878,-178.074,7.237,148.797
C02342=1152.946,198.044,-61.854,-178.076,7.235,148.797
C02343=1152.951,197.794,-61.830,-178.079,7.232,148.797
C02344=1152.956,197.546,-61.806,-178.081,7.230,148.797
C02345=1152.960,197.298,-61.782,-178.085,7.227,148.797
C02346=1152.965,197.049,-61.759,-178.087,7.225,148.798
C02347=1152.970,196.800,-61.734,-178.090,7.223,148.798
C02348=1152.974,196.550,-61.710,-178.092,7.221,148.798
C02349=1152.978,196.302,-61.686,-178.096,7.218,148.798
C02350=1152.983,196.053,-61.663,-178.098,7.216,148.799
C02351=1152.987,195.804,-61.639,-178.101,7.213,148.799
C02352=1152.992,195.555,-61.615,-178.104,7.212,148.799
C02353=1152.996,195.307,-61.591,-178.106,7.209,148.799
C02354=1153.002,195.058,-61.567,-178.109,7.207,148.800
C02355=1153.006,194.809,-61.543,-178.112,7.204,148.800
C02356=1153.011,194.560,-61.520,-178.115,7.202,148.800
C02357=1153.015,194.312,-61.496,-178.117,7.199,148.800
C02358=1153.020,194.063,-61.473,-178.120,7.198,148.801
C02359=1153.024,193.814,-61.448,-178.123,7.195,148.801
C02360=1153.029,193.564,-61.425,-178.126,7.193,148.801
C02361=1153.033,193.315,-61.401,-178.129,7.190,148.801
C02362=1153.038,193.067,-61.377,-178.131,7.188,148.802
C02363=1153.042,192.818,-61.354,-178.134,7.186,148.802
C02364=1153.047,192.570,-61.330,-178.137,7.184,148.802
C02365=1153.051,192.321,-61.307,-178.140,7.181,148.802
C02366=1153.056,192.072,-61.283,-178.143,7.179,148.803
C02367=1153.061,191.823,-61.259,-178.145,7.177,148.803
C02368=1153.065,191.574,-61.236,-178.148,7.175,148.803
C02369=1153.070,191.325,-61.212,-178.150,7.173,148.803
C02370=1153.074,191.077,-61.188,-178.153,7.170,148.804
C02371=1153.079,190.828,-61.165,-178.156,7.168,148.804
C02372=1153.084,190.579,-61.142,-178.159,7.165,148.804
C02373=1153.088,190.330,-61.118,-178.162,7.164,148.804
C02374=1153.093,190.081,-61.094,-178.164,7.161,148.805
C02375=1153.098,189.832,-61.071,-178.167,7.159,148.805
C02376=1153.102,189.583,-61.047,-178.170,7.156,148.805
C02377=1153.107,189.334,-61.024,-178.173,7.154,148.805
C02378=1153.112,189.085,-61.001,-178.175,7.152,148.806
C02379=1153.116,188.837,-60.977,-178.178,7.150,148.806
C02380=1153.121,188.588,-60.953,-178.181,7.148,148.806
C02381=1153.125,188.339,-60.931,-178.184,7.145,148.807
C02382=1153.130,188.091,-60.908,-178.186,7.143,148.807
C02383=1153.135,187.841,-60.884,-178.190,7.141,148.807
C02384=1153.139,187.592,-60.861,-178.192,7.138,148.807
C02385=1153.144,187.343,-60.837,-178.194,7.137,148.808
C02386=1153.148,187.095,-60.813,-178.198,7.134,148.808
C02387=1153.153,186.846,-60.790,-178.200,7.132,148.808
C02388=1153.157,186.597,-60.767,-178.203,7.129,148.808
C02389=1153.162,186.348,-60.744,-178.206,7.128,148.809
C02390=1153.167,186.099,-60.721,-178.209,7.125,148.809
C02391=1153.171,185.850,-60.697,-178.211,7.123,148.809
C02392=1153.176,185.601,-60.674,-178.214,7.121,148.810
C02393=1153.181,185.353,-60.651,-178.217,7.118,148.810
C02394=1153.185,185.104,-60.628,-178.220,7.117,148.810
C02395=1153.190,184.855,-60.605,-178.222,7.114,148.810
C02396=1153.195,184.606,-60.581,-178.225,7.112,148.810
C02397=1153.199,184.357,-60.559,-178.228,7.110,148.811
C02398=1153.204,184.088,-60.534,-178.231,7.108,148.811
C02399=1153.209,183.818,-60.509,-178.234,7.105,148.811
C02400=1153.215,183.548,-60.483,-178.237,7.102,148.812
C02401=1153.219,183.279,-60.458,-178.240,7.100,148.812
C02402=1153.224,183.029,-60.436,-178.243,7.098,148.812
C02403=1153.229,182.780,-60.412,-178.245,7.096,148.812
C02404=1153.232,182.532,-60.390,-178.248,7.094,148.813
C02405=1153.237,182.283,-60.366,-178.251,7.092,148.813
C02406=1153.242,182.034,-60.343,-178.253,7.089,148.813
C02407=1153.246,181.786,-60.320,-178.257,7.087,148.814
C02408=1153.251,181.537,-60.297,-178.259,7.085,148.814
C02409=1153.256,181.287,-60.274,-178.262,7.083,148.814
C02410=1153.260,181.038,-60.252,-178.265,7.080,148.815
C02411=1153.265,180.789,-60.228,-178.268,7.079,148.815
C02412=1153.270,180.541,-60.205,-178.270,7.077,148.815
C02413=1153.274,180.292,-60.183,-178.273,7.074,148.815
C02414=1153.279,180.043,-60.160,-178.276,7.072,148.816
C02415=1153.283,179.794,-60.137,-178.279,7.069,148.816
C02416=1153.288,179.545,-60.114,-178.281,7.068,148.816
C02417=1153.293,179.296,-60.091,-178.284,7.066,148.817
C02418=1153.297,179.047,-60.069,-178.287,7.063,148.817
C02419=1153.302,178.798,-60.045,-178.289,7.061,148.817
C02420=1153.306,178.549,-60.023,-178.292,7.060,148.817
C02421=1153.312,178.300,-60.000,-178.295,7.057,148.818
C02422=1153.316,178.052,-59.978,-178.298,7.055,148.818
C02423=1153.320,177.803,-59.954,-178.301,7.052,148.818
C02424=1153.326,177.554,-59.932,-178.304,7.051,148.819
C02425=1153.330,177.305,-59.909,-178.306,7.049,148.819
C02426=1153.335,177.056,-59.886,-178.309,7.046,148.819
C02427=1153.339,176.807,-59.864,-178.312,7.044,148.819
C02428=1153.344,176.558,-59.841,-178.314,7.042,148.820
C02429=1153.348,176.309,-59.819,-178.317,7.040,148.820
C02430=1153.353,176.060,-59.795,-178.320,7.038,148.820
C02431=1153.358,175.811,-59.774,-178.323,7.036,148.821
C02432=1153.363,175.562,-59.750,-178.326,7.033,148.821
C02433=1153.367,175.313,-59.728,-178.328,7.031,148.821
C02434=1153.371,175.065,-59.706,-178.331,7.030,148.822
C02435=1153.376,174.815,-59.683,-178.334,7.027,148.822
C02436=1153.380,174.566,-59.660,-178.336,7.025,148.822
C02437=1153.386,174.318,-59.638,-178.339,7.023,148.822
C02438=1153.390,174.069,-59.615,-178.342,7.021,148.823
C02439=1153.395,173.819,-59.593,-178.345,7.019,148.823
C02440=1153.400,173.571,-59.570,-178.347,7.017,148.823
C02441=1153.404,173.322,-59.548,-178.351,7.014,148.824
C02442=1153.409,173.073,-59.525,-178.353,7.013,148.824
C02443=1153.413,172.824,-59.503,-178.356,7.011,148.824
C02444=1153.418,172.574,-59.481,-178.359,7.008,148.824
C02445=1153.422,172.326,-59.458,-178.361,7.006,148.825
C02446=1153.427,172.077,-59.436,-178.364,7.004,148.825
C02447=1153.432,171.828,-59.413,-178.367,7.002,148.826
C02448=1153.437,171.579,-59.391,-178.370,7.000,148.826
C02449=1153.441,171.330,-59.369,-178.372,6.998,148.826
C02450=1153.446,171.081,-59.346,-178.375,6.996,148.826
C02451=1153.451,170.832,-59.324,-178.378,6.994,148.827
C02452=1153.455,170.583,-59.302,-178.381,6.992,148.827
C02453=1153.460,170.335,-59.279,-178.383,6.990,148.827
C02454=1153.464,170.085,-59.257,-178.386,6.987,148.828
C02455=1153.469,169.837,-59.235,-178.389,6.986,148.828
C02456=1153.474,169.587,-59.213,-178.392,6.984,148.828
C02457=1153.478,169.338,-59.190,-178.395,6.981,148.829
C02458=1153.483,169.090,-59.168,-178.397,6.979,148.829
C02459=1153.487,168.840,-59.146,-178.400,6.978,148.829
C02460=1153.493,168.591,-59.124,-178.403,6.976,148.830
C02461=1153.497,168.342,-59.102,-178.406,6.973,148.830
C02462=1153.502,168.094,-59.079,-178.408,6.971,148.830
C02463=1153.506,167.845,-59.057,-178.411,6.969,148.831
C02464=1153.511,167.596,-59.036,-178.414,6.967,148.831
C02465=1153.516,167.346,-59.013,-178.417,6.965,148.831
C02466=1153.521,167.098,-58.991,-178.419,6.963,148.831
C02467=1153.525,166.848,-58.969,-178.422,6.961,148.832
C02468=1153.530,166.600,-58.948,-178.425,6.959,148.832
C02469=1153.534,166.351,-58.925,-178.428,6.957,148.832
C02470=1153.540,166.102,-58.903,-178.431,6.955,148.833
C02471=1153.544,165.853,-58.881,-178.433,6.953,148.833
C02472=1153.549,165.604,-58.859,-178.436,6.951,148.833
C02473=1153.553,165.355,-58.837,-178.439,6.949,148.834
C02474=1153.558,165.106,-58.815,-178.441,6.947,148.834
C02475=1153.562,164.857,-58.793,-178.444,6.945,148.834
C02476=1153.567,164.608,-58.771,-178.447,6.943,148.835
C02477=1153.572,164.359,-58.749,-178.450,6.941,148.835
C02478=1153.577,164.110,-58.727,-178.452,6.939,148.835
C02479=1153.581,163.861,-58.705,-178.455,6.937,148.836
C02480=1153.586,163.612,-58.683,-178.458,6.935,148.836
C02481=1153.590,163.363,-58.661,-178.461,6.933,148.836
C02482=1153.595,163.114,-58.640,-178.464,6.931,148.837
C02483=1153.600,162.865,-58.618,-178.466,6.929,148.837
C02484=1153.604,162.616,-58.596,-178.469,6.927,148.837
C02485=1153.609,162.367,-58.574,-178.472,6.925,148.838
C02486=1153.614,162.117,-58.553,-178.475,6.923,148.838
C02487=1153.619,161.869,-58.531,-178.477,6.921,148.838
C02488=1153.623,161.619,-58.509,-178.481,6.919,148.839
C02489=1153.628,161.371,-58.487,-178.483,6.917,148.839
C02490=1153.633,161.122,-58.466,-178.486,6.915,148.839
C02491=1153.637,160.873,-58.444,-178.488,6.913,148.840
C02492=1153.642,160.624,-58.422,-178.492,6.911,148.840
C02493=1153.647,160.375,-58.401,-178.494,6.909,148.840
C02494=1153.651,160.126,-58.379,-178.497,6.907,148.841
C02495=1153.656,159.877,-58.357,-178.499,6.905,148.841
C02496=1153.660,159.628,-58.335,-178.502,6.904,148.841
C02497=1153.665,159.379,-58.314,-178.505,6.901,148.842
C02498=1153.670,159.130,-58.293,-178.508,6.899,148.842
C02499=1153.675,158.880,-58.271,-178.511,6.898,148.842
C02500=1153.680,158.632,-58.249,-178.513,6.896,148.843
C02501=1153.684,158.383,-58.227,-178.517,6.893,148.843
C02502=1153.689,158.114,-58.204,-178.519,6.892,148.844
C02503=1153.695,157.845,-58.181,-178.522,6.890,148.844
C02504=1153.699,157.576,-58.158,-178.525,6.887,148.844
C02505=1153.705,157.307,-58.134,-178.528,6.886,148.845
C02506=1153.710,157.058,-58.113,-178.531,6.883,148.845
C02507=1153.714,156.808,-58.091,-178.533,6.881,148.845
C02508=1153.718,156.560,-58.070,-178.536,6.879,148.846
C02509=1153.723,156.311,-58.049,-178.539,6.877,148.846
C02510=1153.728,156.061,-58.027,-178.542,6.876,148.846
C02511=1153.732,155.813,-58.006,-178.545,6.873,148.847
C02512=1153.738,155.563,-57.985,-178.548,6.871,148.847
C02513=1153.742,155.315,-57.963,-178.550,6.870,148.847
C02514=1153.747,155.065,-57.942,-178.553,6.868,148.848
C02515=1153.751,154.816,-57.920,-178.556,6.866,148.848
C02516=1153.756,154.568,-57.899,-178.558,6.864,148.848
C02517=1153.761,154.319,-57.878,-178.561,6.862,148.849
C02518=1153.765,154.069,-57.856,-178.564,6.860,148.849
C02519=1153.771,153.820,-57.835,-178.567,6.858,148.850
C02520=1153.775,153.572,-57.814,-178.569,6.856,148.850
C02521=1153.780,153.322,-57.793,-178.572,6.855,148.850
C02522=1153.784,153.073,-57.771,-178.575,6.852,148.851
C02523=1153.789,152.824,-57.750,-178.578,6.850,148.851
C02524=1153.794,152.575,-57.729,-178.581,6.849,148.851
C02525=1153.799,152.326,-57.708,-178.583,6.847,148.852
C02526=1153.803,152.076,-57.686,-178.586,6.845,148.852
C02527=1153.808,151.828,-57.665,-178.588,6.843,148.852
C02528=1153.813,151.579,-57.644,-178.591,6.841,148.853
C02529=1153.817,151.330,-57.623,-178.594,6.839,148.853
C02530=1153.823,151.081,-57.602,-178.597,6.837,148.853
C02531=1153.826,150.831,-57.581,-178.600,6.835,148.854
C02532=1153.831,150.582,-57.559,-178.602,6.834,148.854
C02533=1153.837,150.333,-57.538,-178.605,6.832,148.855
C02534=1153.841,150.084,-57.518,-178.608,6.830,148.855
C02535=1153.846,149.836,-57.496,-178.611,6.828,148.855
C02536=1153.851,149.586,-57.475,-178.614,6.826,148.856
C02537=1153.855,149.337,-57.454,-178.616,6.824,148.856
C02538=1153.860,149.088,-57.433,-178.619,6.823,148.856
C02539=1153.865,148.839,-57.412,-178.621,6.820,148.857
C02540=1153.869,148.590,-57.391,-178.624,6.819,148.857
C02541=1153.874,148.341,-57.370,-178.627,6.817,148.857
C02542=1153.879,148.092,-57.349,-178.630,6.815,148.858
C02543=1153.884,147.843,-57.328,-178.633,6.813,148.858
C02544=1153.888,147.593,-57.307,-178.636,6.811,148.859
C02545=1153.893,147.344,-57.287,-178.638,6.809,148.859
C02546=1153.898,147.095,-57.265,-178.641,6.808,148.859
C02547=1153.902,146.847,-57.245,-178.644,6.806,148.860
C02548=1153.907,146.597,-57.224,-178.646,6.804,148.860
C02549=1153.912,146.348,-57.203,-178.649,6.802,148.860
C02550=1153.917,146.099,-57.182,-178.652,6.801,148.861
C02551=1153.922,145.850,-57.161,-178.655,6.798,148.861
C02552=1153.926,145.601,-57.140,-178.658,6.796,148.862
C02553=1153.931,145.352,-57.119,-178.660,6.795,148.862
C02554=1153.936,145.103,-57.099,-178.663,6.793,148.862
C02555=1153.940,144.853,-57.078,-178.666,6.791,148.863
C02556=1153.945,144.604,-57.057,-178.669,6.790,148.863
C02557=1153.950,144.355,-57.036,-178.671,6.788,148.864
C02558=1153.954,144.106,-57.016,-178.674,6.786,148.864
C02559=1153.960,143.857,-56.995,-178.677,6.784,148.864
C02560=1153.964,143.608,-56.975,-178.680,6.781,148.864
C02561=1153.969,143.359,-56.954,-178.682,6.780,148.865
C02562=1153.974,143.110,-56.933,-178.685,6.778,148.865
C02563=1153.978,142.861,-56.913,-178.688,6.776,148.866
C02564=1153.983,142.611,-56.892,-178.690,6.775,148.866
C02565=1153.988,142.363,-56.872,-178.693,6.773,148.866
C02566=1153.993,142.113,-56.851,-178.696,6.771,148.867
C02567=1153.997,141.864,-56.830,-178.698,6.769,148.867
C02568=1154.002,141.615,-56.810,-178.701,6.768,148.868
C02569=1154.007,141.366,-56.789,-178.704,6.766,148.868
C02570=1154.011,141.117,-56.768,-178.707,6.764,148.868
C02571=1154.017,140.868,-56.748,-178.710,6.762,148.869
C02572=1154.021,140.619,-56.727,-178.713,6.760,148.869
C02573=1154.025,140.370,-56.707,-178.715,6.758,148.869
C02574=1154.031,140.121,-56.686,-178.718,6.757,148.870
C02575=1154.035,139.872,-56.665,-178.721,6.755,148.870
C02576=1154.039,139.623,-56.645,-178.723,6.753,148.871
C02577=1154.045,139.373,-56.625,-178.726,6.751,148.871
C02578=1154.049,139.124,-56.604,-178.729,6.750,148.871
C02579=1154.054,138.875,-56.584,-178.732,6.748,148.872
C02580=1154.059,138.626,-56.563,-178.734,6.746,148.872
C02581=1154.063,138.377,-56.543,-178.737,6.745,148.873
C02582=1154.068,138.128,-56.522,-178.740,6.743,148.873
C02583=1154.073,137.878,-56.502,-178.742,6.741,148.873
C02584=1154.078,137.629,-56.482,-178.745,6.739,148.874
C02585=1154.082,137.380,-56.461,-178.748,6.738,148.874
C02586=1154.087,137.132,-56.441,-178.751,6.736,148.875
C02587=1154.093,136.882,-56.421,-178.753,6.734,148.875
C02588=1154.097,136.633,-56.401,-178.757,6.732,148.875
C02589=1154.102,136.384,-56.380,-178.759,6.730,148.876
C02590=1154.106,136.135,-56.360,-178.762,6.728,148.876
C02591=1154.112,135.885,-56.340,-178.765,6.727,148.877
C02592=1154.116,135.636,-56.319,-178.768,6.725,148.877
C02593=1154.120,135.387,-56.299,-178.771,6.723,148.877
C02594=1154.125,135.138,-56.279,-178.773,6.722,148.878
C02595=1154.130,134.890,-56.259,-178.776,6.720,148.878
C02596=1154.135,134.640,-56.238,-178.779,6.718,148.879
C02597=1154.140,134.391,-56.219,-178.781,6.717,148.879
C02598=1154.145,134.142,-56.198,-178.784,6.715,148.879
C02599=1154.149,133.892,-56.179,-178.787,6.713,148.880
C02600=1154.154,133.643,-56.158,-178.790,6.711,148.880
C02601=1154.159,133.394,-56.137,-178.792,6.710,148.881
C02602=1154.164,133.145,-56.118,-178.795,6.708,148.881
C02603=1154.169,132.896,-56.098,-178.798,6.706,148.881
C02604=1154.173,132.647,-56.078,-178.800,6.705,148.882
C02605=1154.178,132.398,-56.058,-178.803,6.703,148.882
C02606=1154.184,132.129,-56.036,-178.806,6.701,148.883
C02607=1154.188,131.860,-56.015,-178.809,6.699,148.883
C02608=1154.193,131.592,-55.993,-178.812,6.697,148.884
C02609=1154.199,131.323,-55.971,-178.815,6.696,148.884
C02610=1154.203,131.074,-55.951,-178.818,6.694,148.884
C02611=1154.208,130.825,-55.932,-178.820,6.692,148.885
C02612=1154.213,130.576,-55.911,-178.823,6.690,148.885
C02613=1154.218,130.327,-55.892,-178.826,6.689,148.886
C02614=1154.222,130.077,-55.872,-178.829,6.687,148.886
C02615=1154.227,129.828,-55.852,-178.831,6.685,148.886
C02616=1154.232,129.579,-55.832,-178.834,6.684,148.887
C02617=1154.237,129.330,-55.812,-178.837,6.682,148.887
C02618=1154.241,129.081,-55.792,-178.839,6.680,148.888
C02619=1154.246,128.831,-55.773,-178.843,6.679,148.888
C02620=1154.251,128.583,-55.753,-178.845,6.677,148.889
C02621=1154.256,128.333,-55.733,-178.848,6.675,148.889
C02622=1154.260,128.085,-55.713,-178.851,6.674,148.889
C02623=1154.265,127.835,-55.693,-178.854,6.672,148.890
C02624=1154.270,127.586,-55.674,-178.856,6.670,148.890
C02625=1154.275,127.337,-55.653,-178.859,6.668,148.891
C02626=1154.280,127.088,-55.634,-178.862,6.667,148.891
C02627=1154.285,126.839,-55.614,-178.864,6.665,148.891
C02628=1154.290,126.589,-55.595,-178.867,6.663,148.892
C02629=1154.294,126.340,-55.574,-178.870,6.662,148.892
C02630=1154.299,126.091,-55.555,-178.873,6.660,148.893
C02631=1154.304,125.842,-55.535,-178.876,6.659,148.893
C02632=1154.309,125.592,-55.516,-178.878,6.657,148.894
C02633=1154.313,125.343,-55.495,-178.881,6.655,148.894
C02634=1154.319,125.094,-55.476,-178.884,6.653,148.894
C02635=1154.323,124.845,-55.456,-178.887,6.652,148.895
C02636=1154.327,124.596,-55.437,-178.889,6.651,148.895
C02637=1154.333,124.347,-55.417,-178.891,6.649,148.896
C02638=1154.337,124.098,-55.398,-178.894,6.647,148.896
C02639=1154.342,123.848,-55.378,-178.897,6.646,148.896
C02640=1154.347,123.599,-55.359,-178.900,6.644,148.897
C02641=1154.352,123.350,-55.339,-178.902,6.642,148.897
C02642=1154.357,123.100,-55.319,-178.905,6.641,148.898
C02643=1154.361,122.852,-55.301,-178.908,6.639,148.898
C02644=1154.366,122.603,-55.280,-178.911,6.637,148.899
C02645=1154.371,122.353,-55.261,-178.914,6.636,148.899
C02646=1154.376,122.104,-55.241,-178.916,6.634,148.899
C02647=1154.381,121.855,-55.222,-178.919,6.632,148.900
C02648=1154.385,121.605,-55.203,-178.922,6.631,148.900
C02649=1154.390,121.357,-55.183,-178.925,6.629,148.901
C02650=1154.395,121.107,-55.164,-178.928,6.628,148.901
C02651=1154.400,120.858,-55.145,-178.930,6.626,148.902
C02652=1154.405,120.609,-55.125,-178.933,6.624,148.902
C02653=1154.409,120.359,-55.106,-178.935,6.623,148.902
C02654=1154.414,120.110,-55.086,-178.938,6.622,148.903
C02655=1154.419,119.861,-55.067,-178.941,6.620,148.903
C02656=1154.424,119.612,-55.048,-178.943,6.618,148.904
C02657=1154.428,119.363,-55.028,-178.946,6.616,148.904
C02658=1154.434,119.114,-55.009,-178.949,6.615,148.905
C02659=1154.438,118.864,-54.990,-178.952,6.613,148.905
C02660=1154.442,118.615,-54.970,-178.955,6.612,148.905
C02661=1154.448,118.366,-54.951,-178.958,6.610,148.906
C02662=1154.453,118.117,-54.932,-178.960,6.608,148.906
C02663=1154.458,117.868,-54.912,-178.963,6.607,148.907
C02664=1154.462,117.618,-54.894,-178.966,6.605,148.907
C02665=1154.468,117.369,-54.875,-178.968,6.604,148.907
C02666=1154.472,117.119,-54.855,-178.971,6.603,148.908
C02667=1154.477,116.871,-54.836,-178.974,6.601,148.908
C02668=1154.482,116.621,-54.817,-178.976,6.599,148.909
C02669=1154.487,116.372,-54.797,-178.979,6.598,148.909
C02670=1154.491,116.123,-54.778,-178.982,6.596,148.910
C02671=1154.497,115.874,-54.760,-178.985,6.594,148.910
C02672=1154.501,115.624,-54.741,-178.988,6.593,148.911
C02673=1154.506,115.376,-54.721,-178.991,6.591,148.911
C02674=1154.511,115.126,-54.702,-178.993,6.590,148.912
C02675=1154.515,114.877,-54.683,-178.995,6.588,148.912
C02676=1154.520,114.627,-54.664,-178.998,6.587,148.912
C02677=1154.525,114.379,-54.645,-179.001,6.585,148.913
C02678=1154.530,114.129,-54.626,-179.004,6.583,148.913
C02679=1154.535,113.880,-54.606,-179.007,6.582,148.914
C02680=1154.539,113.630,-54.588,-179.009,6.580,148.914
C02681=1154.545,113.381,-54.569,-179.012,6.579,148.915
C02682=1154.549,113.132,-54.550,-179.015,6.577,148.915
C02683=1154.554,112.883,-54.531,-179.017,6.576,148.915
C02684=1154.558,112.633,-54.512,-179.020,6.574,148.916
C02685=1154.564,112.385,-54.493,-179.023,6.573,148.916
C02686=1154.569,112.135,-54.475,-179.026,6.571,148.917
C02687=1154.573,111.886,-54.455,-179.028,6.570,148.917
C02688=1154.579,111.637,-54.436,-179.031,6.568,148.918
C02689=1154.583,111.387,-54.417,-179.034,6.566,148.918
C02690=1154.588,111.138,-54.398,-179.036,6.565,148.918
C02691=1154.593,110.889,-54.380,-179.039,6.564,148.919
C02692=1154.597,110.640,-54.361,-179.042,6.562,148.920
C02693=1154.603,110.391,-54.342,-179.045,6.561,148.920
C02694=1154.607,110.141,-54.324,-179.047,6.559,148.920
C02695=1154.612,109.892,-54.304,-179.050,6.557,148.921
C02696=1154.617,109.643,-54.286,-179.053,6.556,148.921
C02697=1154.622,109.393,-54.267,-179.055,6.555,148.922
C02698=1154.627,109.144,-54.249,-179.058,6.553,148.922
C02699=1154.632,108.895,-54.229,-179.061,6.551,148.923
C02700=1154.636,108.646,-54.211,-179.064,6.550,148.923
C02701=1154.641,108.397,-54.192,-179.067,6.548,148.924
C02702=1154.646,108.147,-54.173,-179.070,6.547,148.924
C02703=1154.651,107.898,-54.155,-179.072,6.546,148.924
C02704=1154.656,107.649,-54.136,-179.074,6.544,148.925
C02705=1154.660,107.400,-54.117,-179.077,6.542,148.925
C02706=1154.665,107.150,-54.099,-179.080,6.541,148.926
C02707=1154.671,106.901,-54.080,-179.083,6.539,148.926
C02708=1154.675,106.652,-54.061,-179.086,6.538,148.927
C02709=1154.680,106.402,-54.043,-179.088,6.537,148.927
C02710=1154.685,106.134,-54.023,-179.091,6.535,148.928
C02711=1154.690,105.866,-54.003,-179.094,6.534,148.928
C02712=1154.696,105.597,-53.983,-179.097,6.532,148.929
C02713=1154.700,105.329,-53.963,-179.100,6.530,148.929
C02714=1154.706,105.080,-53.944,-179.102,6.529,148.930
C02715=1154.710,104.830,-53.926,-179.105,6.527,148.930
C02716=1154.715,104.581,-53.907,-179.108,6.526,148.930
C02717=1154.721,104.332,-53.889,-179.111,6.524,148.931
C02718=1154.725,104.082,-53.870,-179.114,6.523,148.932
C02719=1154.730,103.833,-53.852,-179.116,6.522,148.932
C02720=1154.735,103.584,-53.834,-179.119,6.520,148.932
C02721=1154.740,103.335,-53.815,-179.121,6.518,148.933
C02722=1154.744,103.085,-53.797,-179.125,6.517,148.933
C02723=1154.749,102.836,-53.778,-179.127,6.515,148.934
C02724=1154.754,102.587,-53.760,-179.129,6.514,148.934
C02725=1154.760,102.338,-53.741,-179.132,6.513,148.935
C02726=1154.764,102.088,-53.723,-179.135,6.511,148.935
C02727=1154.769,101.839,-53.704,-179.138,6.510,148.936
C02728=1154.773,101.590,-53.686,-179.141,6.508,148.936
C02729=1154.779,101.341,-53.668,-179.143,6.507,148.937
C02730=1154.783,101.091,-53.649,-179.146,6.505,148.937
C02731=1154.788,100.842,-53.631,-179.149,6.504,148.938
C02732=1154.793,100.593,-53.613,-179.152,6.502,148.938
C02733=1154.798,100.344,-53.595,-179.154,6.502,148.938
C02734=1154.803,100.095,-53.577,-179.157,6.500,148.939
C02735=1154.808,99.844,-53.558,-179.160,6.499,148.939
C02736=1154.813,99.595,-53.540,-179.162,6.497,148.940
C02737=1154.818,99.346,-53.522,-179.165,6.495,148.940
C02738=1154.823,99.097,-53.504,-179.167,6.494,148.941
C02739=1154.827,98.848,-53.486,-179.171,6.493,148.941
C02740=1154.831,98.599,-53.467,-179.173,6.491,148.942
C02741=1154.836,98.349,-53.449,-179.176,6.490,148.942
C02742=1154.842,98.100,-53.430,-179.178,6.489,148.943
C02743=1154.847,97.851,-53.412,-179.181,6.487,148.943
C02744=1154.852,97.602,-53.394,-179.184,6.486,148.944
C02745=1154.857,97.352,-53.376,-179.187,6.484,148.944
C02746=1154.861,97.102,-53.358,-179.189,6.483,148.944
C02747=1154.866,96.853,-53.340,-179.192,6.482,148.945
C02748=1154.871,96.604,-53.322,-179.195,6.480,148.946
C02749=1154.876,96.355,-53.304,-179.198,6.478,148.946
C02750=1154.881,96.106,-53.286,-179.200,6.477,148.946
C02751=1154.886,95.857,-53.268,-179.203,6.476,148.947
C02752=1154.891,95.607,-53.250,-179.206,6.474,148.947
C02753=1154.895,95.358,-53.232,-179.208,6.473,148.948
C02754=1154.900,95.108,-53.214,-179.211,6.472,148.948
C02755=1154.905,94.859,-53.196,-179.214,6.471,148.949
C02756=1154.910,94.609,-53.179,-179.217,6.469,148.949
C02757=1154.915,94.360,-53.161,-179.219,6.467,148.950
C02758=1154.920,94.111,-53.143,-179.221,6.466,148.950
C02759=1154.925,93.862,-53.125,-179.225,6.465,148.951
C02760=1154.930,93.613,-53.107,-179.227,6.463,148.951
C02761=1154.934,93.364,-53.089,-179.230,6.462,148.952
C02762=1154.939,93.114,-53.071,-179.232,6.461,148.952
C02763=1154.944,92.865,-53.053,-179.235,6.459,148.953
C02764=1154.949,92.615,-53.035,-179.238,6.458,148.953
C02765=1154.954,92.365,-53.017,-179.240,6.457,148.954
C02766=1154.959,92.116,-52.999,-179.243,6.455,148.954
C02767=1154.964,91.867,-52.981,-179.246,6.454,148.955
C02768=1154.969,91.618,-52.963,-179.249,6.452,148.955
C02769=1154.974,91.368,-52.946,-179.251,6.451,148.955
C02770=1154.979,91.119,-52.928,-179.254,6.450,148.956
C02771=1154.984,90.870,-52.910,-179.257,6.448,148.957
C02772=1154.989,90.621,-52.892,-179.259,6.447,148.957
C02773=1154.994,90.371,-52.875,-179.262,6.446,148.958
C02774=1154.998,90.122,-52.857,-179.265,6.444,148.958
C02775=1155.003,89.873,-52.839,-179.268,6.443,148.958
C02776=1155.008,89.624,-52.821,-179.270,6.442,148.959
C02777=1155.013,89.374,-52.804,-179.273,6.440,148.960
C02778=1155.018,89.125,-52.786,-179.276,6.439,148.960
C02779=1155.023,88.875,-52.768,-179.278,6.438,148.960
C02780=1155.028,88.626,-52.751,-179.281,6.437,148.961
C02781=1155.032,88.377,-52.734,-179.284,6.435,148.961
C02782=1155.037,88.128,-52.716,-179.286,6.434,148.962
C02783=1155.042,87.878,-52.698,-179.289,6.432,148.962
C02784=1155.047,87.629,-52.680,-179.292,6.431,148.963
C02785=1155.052,87.379,-52.662,-179.294,6.430,148.963
C02786=1155.057,87.130,-52.646,-179.297,6.428,148.964
C02787=1155.062,86.881,-52.628,-179.300,6.427,148.964
C02788=1155.067,86.631,-52.610,-179.303,6.425,148.965
C02789=1155.072,86.382,-52.592,-179.305,6.425,148.965
C02790=1155.077,86.133,-52.574,-179.308,6.423,148.966
C02791=1155.081,85.883,-52.558,-179.311,6.422,148.966
C02792=1155.086,85.634,-52.540,-179.313,6.421,148.967
C02793=1155.091,85.384,-52.523,-179.316,6.419,148.967
C02794=1155.097,85.136,-52.505,-179.319,6.418,148.968
C02795=1155.101,84.886,-52.488,-179.321,6.417,148.968
C02796=1155.106,84.637,-52.470,-179.324,6.415,148.969
C02797=1155.111,84.387,-52.453,-179.327,6.414,148.969
C02798=1155.115,84.138,-52.436,-179.329,6.413,148.970
C02799=1155.121,83.889,-52.418,-179.332,6.411,148.970
C02800=1155.126,83.639,-52.400,-179.335,6.410,148.971
C02801=1155.131,83.390,-52.383,-179.337,6.409,148.971
C02802=1155.135,83.141,-52.366,-179.340,6.407,148.972
C02803=1155.140,82.891,-52.348,-179.343,6.406,148.972
C02804=1155.145,82.641,-52.331,-179.346,6.405,148.973
C02805=1155.150,82.393,-52.314,-179.348,6.404,148.973
C02806=1155.155,82.143,-52.297,-179.352,6.402,148.974
C02807=1155.160,81.894,-52.279,-179.354,6.401,148.974
C02808=1155.165,81.645,-52.262,-179.356,6.400,148.975
C02809=1155.170,81.395,-52.245,-179.359,6.399,148.975
C02810=1155.175,81.146,-52.227,-179.362,6.397,148.976
C02811=1155.179,80.896,-52.210,-179.364,6.396,148.976
C02812=1155.185,80.647,-52.193,-179.367,6.395,148.977
C02813=1155.189,80.398,-52.176,-179.370,6.394,148.977
C02814=1155.195,80.129,-52.157,-179.373,6.392,148.978
C02815=1155.200,79.860,-52.139,-179.376,6.391,148.978
C02816=1155.205,79.593,-52.121,-179.379,6.389,148.979
C02817=1155.211,79.324,-52.102,-179.381,6.388,148.979
C02818=1155.216,79.075,-52.084,-179.384,6.387,148.980
C02819=1155.220,78.825,-52.068,-179.387,6.385,148.980
C02820=1155.226,78.576,-52.051,-179.389,6.385,148.981
C02821=1155.230,78.327,-52.033,-179.392,6.383,148.981
C02822=1155.235,78.077,-52.016,-179.395,6.382,148.982
C02823=1155.240,77.828,-51.999,-179.397,6.381,148.982
C02824=1155.245,77.578,-51.982,-179.400,6.379,148.983
C02825=1155.250,77.330,-51.965,-179.403,6.378,148.984
C02826=1155.255,77.080,-51.948,-179.405,6.377,148.984
C02827=1155.260,76.830,-51.931,-179.408,6.375,148.984
C02828=1155.265,76.581,-51.914,-179.411,6.375,148.985
C02829=1155.271,76.332,-51.897,-179.414,6.373,148.985
C02830=1155.275,76.082,-51.880,-179.416,6.372,148.986
C02831=1155.279,75.833,-51.863,-179.419,6.371,148.987
C02832=1155.285,75.584,-51.846,-179.422,6.369,148.987
C02833=1155.289,75.334,-51.829,-179.424,6.368,148.987
C02834=1155.295,75.085,-51.812,-179.427,6.367,148.988
C02835=1155.299,74.835,-51.795,-179.429,6.366,148.988
C02836=1155.305,74.586,-51.778,-179.432,6.364,148.989
C02837=1155.310,74.337,-51.762,-179.435,6.363,148.990
C02838=1155.315,74.087,-51.745,-179.437,6.362,148.990
C02839=1155.319,73.838,-51.728,-179.440,6.361,148.990
C02840=1155.324,73.588,-51.710,-179.443,6.360,148.991
C02841=1155.329,73.340,-51.694,-179.445,6.358,148.991
C02842=1155.334,73.090,-51.677,-179.448,6.357,148.992
C02843=1155.339,72.840,-51.660,-179.451,6.356,148.993
C02844=1155.343,72.591,-51.643,-179.454,6.354,148.993
C02845=1155.349,72.342,-51.626,-179.456,6.354,148.994
C02846=1155.354,72.092,-51.610,-179.459,6.352,148.994
C02847=1155.358,71.843,-51.593,-179.461,6.351,148.995
C02848=1155.364,71.594,-51.576,-179.464,6.350,148.995
C02849=1155.369,71.344,-51.559,-179.467,6.348,148.996
C02850=1155.373,71.095,-51.543,-179.469,6.348,148.996
C02851=1155.379,70.846,-51.526,-179.472,6.346,148.997
C02852=1155.384,70.596,-51.510,-179.475,6.345,148.997
C02853=1155.388,70.346,-51.493,-179.478,6.344,148.998
C02854=1155.394,70.097,-51.476,-179.480,6.343,148.998
C02855=1155.398,69.848,-51.460,-179.483,6.342,148.999
C02856=1155.403,69.598,-51.443,-179.486,6.340,148.999
C02857=1155.409,69.349,-51.426,-179.488,6.339,149.000
C02858=1155.413,69.099,-51.409,-179.491,6.338,149.000
C02859=1155.418,68.850,-51.393,-179.493,6.337,149.001
C02860=1155.423,68.601,-51.376,-179.496,6.336,149.001
C02861=1155.428,68.351,-51.359,-179.498,6.335,149.002
C02862=1155.433,68.102,-51.343,-179.501,6.333,149.002
C02863=1155.438,67.852,-51.327,-179.504,6.333,149.003
C02864=1155.443,67.603,-51.310,-179.507,6.331,149.003
C02865=1155.448,67.354,-51.293,-179.510,6.330,149.004
C02866=1155.453,67.104,-51.277,-179.512,6.329,149.004
C02867=1155.458,66.855,-51.261,-179.515,6.327,149.005
C02868=1155.463,66.605,-51.244,-179.517,6.327,149.005
C02869=1155.468,66.356,-51.227,-179.520,6.325,149.006
C02870=1155.473,66.107,-51.211,-179.523,6.324,149.007
C02871=1155.477,65.857,-51.194,-179.525,6.323,149.007
C02872=1155.483,65.608,-51.178,-179.528,6.322,149.008
C02873=1155.488,65.358,-51.161,-179.531,6.321,149.008
C02874=1155.492,65.109,-51.145,-179.533,6.320,149.008
C02875=1155.497,64.860,-51.128,-179.536,6.318,149.009
C02876=1155.502,64.610,-51.112,-179.538,6.318,149.010
C02877=1155.507,64.361,-51.096,-179.541,6.316,149.010
C02878=1155.512,64.112,-51.079,-179.544,6.315,149.011
C02879=1155.518,63.862,-51.063,-179.546,6.314,149.011
C02880=1155.522,63.612,-51.046,-179.550,6.312,149.012
C02881=1155.527,63.364,-51.030,-179.552,6.312,149.012
C02882=1155.532,63.114,-51.014,-179.555,6.310,149.013
C02883=1155.537,62.864,-50.998,-179.557,6.309,149.013
C02884=1155.542,62.615,-50.981,-179.560,6.308,149.014
C02885=1155.547,62.365,-50.965,-179.562,6.307,149.014
C02886=1155.552,62.116,-50.949,-179.565,6.306,149.015
C02887=1155.557,61.866,-50.932,-179.568,6.305,149.016
C02888=1155.562,61.617,-50.916,-179.571,6.303,149.016
C02889=1155.567,61.368,-50.899,-179.573,6.303,149.016
C02890=1155.572,61.118,-50.884,-179.576,6.301,149.017
C02891=1155.577,60.869,-50.867,-179.578,6.300,149.017
C02892=1155.582,60.619,-50.852,-179.581,6.299,149.018
C02893=1155.586,60.370,-50.835,-179.583,6.298,149.019
C02894=1155.592,60.121,-50.819,-179.586,6.297,149.019
C02895=1155.596,59.871,-50.803,-179.589,6.296,149.020
C02896=1155.602,59.622,-50.787,-179.592,6.294,149.020
C02897=1155.606,59.372,-50.770,-179.594,6.294,149.021
C02898=1155.612,59.123,-50.755,-179.597,6.292,149.021
C02899=1155.617,58.874,-50.739,-179.599,6.291,149.022
C02900=1155.621,58.624,-50.723,-179.602,6.290,149.022
C02901=1155.627,58.375,-50.706,-179.604,6.289,149.023
C02902=1155.631,58.125,-50.690,-179.608,6.288,149.023
C02903=1155.636,57.876,-50.674,-179.610,6.287,149.024
C02904=1155.641,57.626,-50.658,-179.613,6.285,149.024
C02905=1155.646,57.377,-50.642,-179.615,6.285,149.025
C02906=1155.651,57.127,-50.626,-179.617,6.284,149.025
C02907=1155.656,56.878,-50.610,-179.621,6.283,149.026
C02908=1155.662,56.629,-50.594,-179.623,6.282,149.027
C02909=1155.666,56.379,-50.578,-179.626,6.281,149.027
C02910=1155.671,56.130,-50.562,-179.628,6.280,149.028
C02911=1155.676,55.880,-50.546,-179.631,6.278,149.028
C02912=1155.682,55.631,-50.530,-179.634,6.278,149.029
C02913=1155.687,55.382,-50.514,-179.636,6.276,149.029
C02914=1155.691,55.132,-50.498,-179.639,6.275,149.030
C02915=1155.697,54.882,-50.482,-179.642,6.274,149.030
C02916=1155.701,54.633,-50.466,-179.644,6.273,149.031
C02917=1155.707,54.383,-50.450,-179.647,6.272,149.031
C02918=1155.712,54.115,-50.433,-179.650,6.271,149.032
C02919=1155.718,53.847,-50.416,-179.652,6.269,149.032
C02920=1155.723,53.577,-50.399,-179.656,6.268,149.033
C02921=1155.728,53.309,-50.382,-179.658,6.267,149.034
C02922=1155.733,53.060,-50.367,-179.661,6.266,149.034
C02923=1155.738,52.811,-50.350,-179.663,6.265,149.035
C02924=1155.743,52.561,-50.334,-179.666,6.264,149.035
C02925=1155.748,52.311,-50.319,-179.669,6.263,149.036
C02926=1155.754,52.062,-50.303,-179.671,6.262,149.036
C02927=1155.758,51.813,-50.286,-179.674,6.261,149.037
C02928=1155.763,51.564,-50.271,-179.676,6.260,149.037
C02929=1155.768,51.314,-50.256,-179.679,6.259,149.038
C02930=1155.773,51.064,-50.240,-179.682,6.258,149.038
C02931=1155.778,50.815,-50.224,-179.685,6.257,149.039
C02932=1155.784,50.565,-50.209,-179.687,6.256,149.040
C02933=1155.787,50.316,-50.193,-179.690,6.255,149.040
C02934=1155.793,50.067,-50.177,-179.692,6.254,149.041
C02935=1155.798,49.817,-50.162,-179.694,6.253,149.041
C02936=1155.803,49.567,-50.146,-179.698,6.252,149.042
C02937=1155.808,49.318,-50.130,-179.700,6.251,149.042
C02938=1155.813,49.069,-50.115,-179.703,6.249,149.043
C02939=1155.818,48.819,-50.099,-179.705,6.249,149.043
C02940=1155.823,48.569,-50.083,-179.708,6.248,149.044
C02941=1155.828,48.321,-50.068,-179.711,6.246,149.044
C02942=1155.833,48.071,-50.052,-179.713,6.246,149.045
C02943=1155.838,47.821,-50.036,-179.716,6.244,149.046
C02944=1155.843,47.572,-50.021,-179.718,6.243,149.046
C02945=1155.848,47.323,-50.006,-179.721,6.242,149.047
C02946=1155.853,47.073,-49.990,-179.724,6.241,149.047
C02947=1155.858,46.823,-49.974,-179.726,6.241,149.048
C02948=1155.863,46.574,-49.959,-179.729,6.239,149.048
C02949=1155.868,46.325,-49.943,-179.732,6.239,149.049
C02950=1155.873,46.075,-49.928,-179.734,6.237,149.049
C02951=1155.878,45.825,-49.912,-179.737,6.236,149.050
C02952=1155.883,45.576,-49.897,-179.739,6.236,149.050
C02953=1155.888,45.327,-49.881,-179.742,6.234,149.051
C02954=1155.894,45.077,-49.866,-179.745,6.234,149.052
C02955=1155.898,44.827,-49.850,-179.747,6.232,149.052
C02956=1155.903,44.578,-49.835,-179.750,6.231,149.053
C02957=1155.908,44.329,-49.820,-179.752,6.231,149.053
C02958=1155.913,44.080,-49.804,-179.755,6.229,149.054
C02959=1155.919,43.830,-49.789,-179.757,6.228,149.054
C02960=1155.923,43.580,-49.774,-179.761,6.227,149.055
C02961=1155.928,43.330,-49.758,-179.763,6.226,149.055
C02962=1155.934,43.081,-49.743,-179.765,6.225,149.056
C02963=1155.938,42.832,-49.728,-179.768,6.224,149.057
C02964=1155.944,42.582,-49.712,-179.770,6.223,149.057
C02965=1155.948,42.333,-49.697,-179.773,6.223,149.058
C02966=1155.953,42.083,-49.681,-179.776,6.221,149.058
C02967=1155.958,41.834,-49.667,-179.778,6.221,149.059
C02968=1155.963,41.584,-49.651,-179.781,6.219,149.059
C02969=1155.969,41.335,-49.636,-179.784,6.219,149.060
C02970=1155.973,41.086,-49.621,-179.786,6.218,149.060
C02971=1155.979,40.836,-49.605,-179.789,6.216,149.061
C02972=1155.983,40.587,-49.590,-179.791,6.216,149.061
C02973=1155.989,40.336,-49.575,-179.794,6.215,149.062
C02974=1155.993,40.087,-49.560,-179.797,6.213,149.063
C02975=1155.999,39.838,-49.544,-179.799,6.213,149.063
C02976=1156.003,39.589,-49.529,-179.802,6.212,149.064
C02977=1156.009,39.339,-49.515,-179.804,6.210,149.064
C02978=1156.014,39.090,-49.500,-179.807,6.210,149.065
C02979=1156.019,38.840,-49.484,-179.810,6.208,149.065
C02980=1156.024,38.591,-49.469,-179.812,6.208,149.066
C02981=1156.029,38.341,-49.454,-179.815,6.207,149.066
C02982=1156.033,38.091,-49.439,-179.818,6.206,149.067
C02983=1156.039,37.842,-49.423,-179.820,6.205,149.067
C02984=1156.044,37.592,-49.409,-179.823,6.204,149.068
C02985=1156.049,37.343,-49.393,-179.825,6.203,149.069
C02986=1156.054,37.094,-49.378,-179.828,6.202,149.069
C02987=1156.059,36.844,-49.363,-179.830,6.201,149.070
C02988=1156.064,36.595,-49.348,-179.833,6.200,149.070
C02989=1156.069,36.345,-49.333,-179.836,6.199,149.071
C02990=1156.074,36.096,-49.319,-179.838,6.199,149.071
C02991=1156.079,35.847,-49.304,-179.841,6.197,149.072
C02992=1156.085,35.596,-49.289,-179.843,6.196,149.072
C02993=1156.089,35.347,-49.274,-179.846,6.196,149.073
C02994=1156.095,35.098,-49.258,-179.849,6.194,149.074
C02995=1156.100,34.848,-49.244,-179.851,6.194,149.074
C02996=1156.104,34.599,-49.229,-179.853,6.193,149.075
C02997=1156.109,34.348,-49.214,-179.857,6.192,149.075
C02998=1156.114,34.099,-49.199,-179.859,6.191,149.076
C02999=1156.120,33.849,-49.184,-179.861,6.190,149.076
C03000=1156.124,33.600,-49.169,-179.864,6.189,149.077
C03001=1156.129,33.351,-49.154,-179.867,6.188,149.078
C03002=1156.135,33.101,-49.139,-179.869,6.187,149.078
C03003=1156.139,32.852,-49.124,-179.872,6.186,149.079
C03004=1156.144,32.602,-49.110,-179.874,6.185,149.079
C03005=1156.150,32.353,-49.094,-179.877,6.184,149.080
C03006=1156.155,32.103,-49.080,-179.880,6.183,149.080
C03007=1156.160,31.854,-49.066,-179.882,6.182,149.081
C03008=1156.165,31.604,-49.050,-179.885,6.182,149.081
C03009=1156.170,31.354,-49.036,-179.887,6.181,149.082
C03010=1156.175,31.105,-49.021,-179.890,6.180,149.083
C03011=1156.180,30.856,-49.006,-179.892,6.179,149.083
C03012=1156.185,30.606,-48.991,-179.895,6.178,149.084
C03013=1156.191,30.357,-48.977,-179.898,6.177,149.084
C03014=1156.195,30.108,-48.962,-179.900,6.176,149.085
C03015=1156.201,29.858,-48.947,-179.902,6.175,149.085
C03016=1156.206,29.608,-48.933,-179.906,6.174,149.086
C03017=1156.211,29.359,-48.918,-179.908,6.173,149.086
C03018=1156.215,29.110,-48.903,-179.910,6.173,149.087
C03019=1156.221,28.860,-48.889,-179.913,6.172,149.088
C03020=1156.226,28.610,-48.874,-179.916,6.171,149.088
C03021=1156.231,28.361,-48.859,-179.918,6.170,149.089
C03022=1156.236,28.092,-48.844,-179.921,6.170,149.089
C03023=1156.242,27.823,-48.827,-179.924,6.168,149.090
C03024=1156.247,27.554,-48.812,-179.926,6.167,149.090
C03025=1156.252,27.285,-48.796,-179.929,6.166,149.091
C03026=1156.257,27.036,-48.782,-179.931,6.165,149.092
C03027=1156.263,26.786,-48.767,-179.934,6.165,149.092
C03028=1156.268,26.537,-48.753,-179.937,6.163,149.093
C03029=1156.273,26.287,-48.738,-179.939,6.163,149.093
C03030=1156.278,26.038,-48.724,-179.942,6.162,149.094
C03031=1156.283,25.788,-48.709,-179.945,6.161,149.095
C03032=1156.288,25.538,-48.694,-179.947,6.160,149.095
C03033=1156.293,25.289,-48.679,-179.950,6.159,149.096
C03034=1156.298,25.039,-48.665,-179.952,6.158,149.096
C03035=1156.303,24.789,-48.651,-179.955,6.157,149.097
C03036=1156.309,24.540,-48.637,-179.957,6.156,149.097
C03037=1156.313,24.291,-48.622,-179.960,6.156,149.098
C03038=1156.318,24.042,-48.608,-179.962,6.155,149.098
C03039=1156.323,23.792,-48.593,-179.965,6.154,149.099
C03040=1156.329,23.542,-48.579,-179.967,6.153,149.100
C03041=1156.334,23.292,-48.564,-179.970,6.153,149.100
C03042=1156.339,23.042,-48.550,-179.972,6.152,149.101
C03043=1156.344,22.794,-48.535,-179.976,6.150,149.101
C03044=1156.349,22.544,-48.521,-179.978,6.150,149.102
C03045=1156.354,22.295,-48.507,-179.980,6.149,149.102
C03046=1156.359,22.045,-48.493,-179.983,6.148,149.103
C03047=1156.364,21.795,-48.478,-179.986,6.147,149.104
C03048=1156.369,21.546,-48.464,-179.988,6.146,149.104
C03049=1156.374,21.297,-48.450,-179.991,6.146,149.105
C03050=1156.379,21.047,-48.436,-179.993,6.145,149.105
C03051=1156.384,20.797,-48.422,-179.996,6.144,149.106
C03052=1156.389,20.547,-48.407,-179.998,6.143,149.106
C03053=1156.394,20.298,-48.392,179.999,6.142,149.107
C03054=1156.399,20.049,-48.378,179.997,6.142,149.107
C03055=1156.404,19.800,-48.364,179.994,6.140,149.108
C03056=1156.409,19.550,-48.350,179.992,6.139,149.109
C03057=1156.414,19.300,-48.336,179.989,6.139,149.109
C03058=1156.419,19.050,-48.321,179.987,6.138,149.110
C03059=1156.425,18.801,-48.307,179.984,6.138,149.110
C03060=1156.430,18.552,-48.293,179.981,6.136,149.111
C03061=1156.435,18.302,-48.279,179.979,6.136,149.112
C03062=1156.440,18.052,-48.265,179.977,6.135,149.112
C03063=1156.445,17.803,-48.251,179.974,6.134,149.113
C03064=1156.450,17.554,-48.236,179.971,6.133,149.113
C03065=1156.455,17.304,-48.222,179.969,6.132,149.114
C03066=1156.460,17.054,-48.208,179.966,6.131,149.114
C03067=1156.466,16.805,-48.195,179.964,6.131,149.115
C03068=1156.471,16.555,-48.180,179.962,6.130,149.115
C03069=1156.476,16.305,-48.166,179.958,6.129,149.116
C03070=1156.481,16.055,-48.152,179.956,6.128,149.117
C03071=1156.486,15.806,-48.138,179.953,6.128,149.117
C03072=1156.491,15.557,-48.124,179.951,6.127,149.118
C03073=1156.496,15.307,-48.109,179.949,6.126,149.118
C03074=1156.501,15.058,-48.096,179.946,6.125,149.119
C03075=1156.506,14.809,-48.082,179.943,6.124,149.120
C03076=1156.511,14.558,-48.068,179.941,6.123,149.120
C03077=1156.516,14.309,-48.054,179.938,6.123,149.121
C03078=1156.522,14.060,-48.040,179.936,6.121,149.121
C03079=1156.527,13.810,-48.026,179.933,6.121,149.122
C03080=1156.532,13.560,-48.011,179.931,6.120,149.122
C03081=1156.537,13.311,-47.997,179.928,6.119,149.123
C03082=1156.542,13.061,-47.984,179.926,6.119,149.123
C03083=1156.547,12.811,-47.970,179.923,6.118,149.124
C03084=1156.552,12.562,-47.956,179.921,6.117,149.125
C03085=1156.557,12.313,-47.942,179.918,6.116,149.125
C03086=1156.563,12.062,-47.928,179.916,6.115,149.126
C03087=1156.568,11.813,-47.915,179.913,6.115,149.126
C03088=1156.572,11.564,-47.901,179.911,6.114,149.127
C03089=1156.577,11.314,-47.887,179.908,6.113,149.128
C03090=1156.583,11.065,-47.873,179.906,6.112,149.128
C03091=1156.588,10.815,-47.859,179.903,6.111,149.129
C03092=1156.592,10.565,-47.845,179.901,6.111,149.129
C03093=1156.598,10.316,-47.832,179.898,6.110,149.130
C03094=1156.603,10.066,-47.818,179.896,6.109,149.130
C03095=1156.609,9.817,-47.804,179.893,6.108,149.131
C03096=1156.614,9.567,-47.790,179.890,6.107,149.131
C03097=1156.618,9.317,-47.777,179.888,6.107,149.132
C03098=1156.624,9.068,-47.763,179.886,6.106,149.133
C03099=1156.629,8.819,-47.749,179.883,6.106,149.133
C03100=1156.634,8.569,-47.735,179.881,6.105,149.134
C03101=1156.639,8.320,-47.722,179.878,6.103,149.134
C03102=1156.644,8.070,-47.707,179.875,6.103,149.135
C03103=1156.650,7.820,-47.694,179.873,6.102,149.136
C03104=1156.654,7.571,-47.681,179.870,6.102,149.136
C03105=1156.660,7.321,-47.667,179.868,6.101,149.137
C03106=1156.665,7.072,-47.653,179.865,6.100,149.137
C03107=1156.670,6.822,-47.639,179.863,6.099,149.138
C03108=1156.675,6.573,-47.626,179.860,6.098,149.139
C03109=1156.680,6.323,-47.612,179.858,6.098,149.139
C03110=1156.685,6.073,-47.599,179.855,6.097,149.140
C03111=1156.690,5.824,-47.585,179.853,6.096,149.140
C03112=1156.696,5.574,-47.572,179.850,6.096,149.141
C03113=1156.700,5.324,-47.558,179.848,6.095,149.141
C03114=1156.705,5.074,-47.545,179.845,6.094,149.142
C03115=1156.711,4.825,-47.531,179.843,6.093,149.142
C03116=1156.715,4.576,-47.517,179.840,6.093,149.143
C03117=1156.721,4.326,-47.504,179.838,6.092,149.144
C03118=1156.726,4.077,-47.490,179.835,6.091,149.144
C03119=1156.731,3.827,-47.477,179.833,6.090,149.145
C03120=1156.736,3.577,-47.463,179.830,6.090,149.145
C03121=1156.742,3.328,-47.450,179.828,6.088,149.146
C03122=1156.746,3.078,-47.437,179.825,6.088,149.147
C03123=1156.752,2.829,-47.423,179.823,6.087,149.147
C03124=1156.756,2.579,-47.410,179.820,6.087,149.148
C03125=1156.762,2.330,-47.396,179.818,6.086,149.148
C03126=1156.767,2.060,-47.381,179.815,6.085,149.149
C03127=1156.772,1.791,-47.367,179.812,6.084,149.150
C03128=1156.778,1.521,-47.352,179.810,6.083,149.150
C03129=1156.784,1.252,-47.338,179.807,6.083,149.151
C03130=1156.789,1.002,-47.324,179.804,6.082,149.151
C03131=1156.794,0.753,-47.311,179.802,6.082,149.152
C03132=1156.799,0.503,-47.298,179.799,6.080,149.153
C03133=1156.804,0.254,-47.284,179.797,6.080,149.153
C03134=1156.809,0.004,-47.271,179.794,6.079,149.154
C03135=1156.814,-0.246,-47.258,179.792,6.078,149.154
C03136=1156.819,-0.495,-47.244,179.789,6.078,149.155
C03137=1156.825,-0.745,-47.231,179.787,6.077,149.155
C03138=1156.830,-0.994,-47.218,179.785,6.077,149.156
C03139=1156.835,-1.244,-47.205,179.782,6.076,149.156
C03140=1156.840,-1.493,-47.191,179.780,6.075,149.157
C03141=1156.845,-1.743,-47.178,179.777,6.074,149.158
C03142=1156.851,-1.992,-47.164,179.774,6.073,149.158
C03143=1156.855,-2.242,-47.151,179.772,6.072,149.159
C03144=1156.861,-2.492,-47.138,179.770,6.072,149.159
C03145=1156.866,-2.741,-47.126,179.767,6.071,149.160
C03146=1156.871,-2.991,-47.111,179.765,6.071,149.161
C03147=1156.876,-3.240,-47.099,179.762,6.070,149.161
C03148=1156.881,-3.490,-47.086,179.760,6.069,149.162
C03149=1156.887,-3.740,-47.073,179.757,6.069,149.162
C03150=1156.891,-3.989,-47.059,179.755,6.068,149.163
C03151=1156.897,-4.239,-47.046,179.752,6.067,149.164
C03152=1156.902,-4.488,-47.033,179.750,6.066,149.164
C03153=1156.907,-4.739,-47.020,179.747,6.066,149.165
C03154=1156.912,-4.988,-47.007,179.745,6.065,149.165
C03155=1156.916,-5.237,-46.993,179.742,6.064,149.166
C03156=1156.922,-5.487,-46.980,179.740,6.064,149.166
C03157=1156.927,-5.736,-46.968,179.737,6.063,149.167
C03158=1156.933,-5.987,-46.954,179.735,6.062,149.168
C03159=1156.938,-6.236,-46.941,179.732,6.062,149.168
C03160=1156.943,-6.485,-46.929,179.730,6.061,149.169
C03161=1156.948,-6.736,-46.915,179.728,6.061,149.169
C03162=1156.953,-6.984,-46.902,179.725,6.060,149.170
C03163=1156.958,-7.234,-46.889,179.723,6.059,149.171
C03164=1156.963,-7.484,-46.876,179.720,6.058,149.171
C03165=1156.968,-7.733,-46.863,179.717,6.057,149.172
C03166=1156.974,-7.983,-46.850,179.715,6.057,149.172
C03167=1156.979,-8.233,-46.837,179.713,6.056,149.173
C03168=1156.984,-8.482,-46.824,179.710,6.055,149.173
C03169=1156.989,-8.732,-46.812,179.708,6.055,149.174
C03170=1156.994,-8.982,-46.798,179.705,6.054,149.175
C03171=1156.999,-9.231,-46.786,179.703,6.054,149.175
C03172=1157.005,-9.480,-46.773,179.701,6.053,149.176
C03173=1157.010,-9.731,-46.759,179.698,6.052,149.176
C03174=1157.015,-9.980,-46.747,179.695,6.052,149.177
C03175=1157.020,-10.229,-46.734,179.693,6.051,149.178
C03176=1157.025,-10.480,-46.721,179.691,6.051,149.178
C03177=1157.030,-10.729,-46.708,179.688,6.050,149.179
C03178=1157.036,-10.978,-46.695,179.686,6.049,149.179
C03179=1157.040,-11.228,-46.682,179.684,6.049,149.180
C03180=1157.046,-11.478,-46.669,179.681,6.048,149.181
C03181=1157.051,-11.727,-46.657,179.679,6.047,149.181
C03182=1157.056,-11.977,-46.644,179.676,6.047,149.182
C03183=1157.061,-12.227,-46.631,179.673,6.045,149.182
C03184=1157.067,-12.476,-46.618,179.671,6.045,149.183
C03185=1157.072,-12.726,-46.605,179.668,6.044,149.183
C03186=1157.076,-12.976,-46.592,179.666,6.044,149.184
C03187=1157.081,-13.225,-46.580,179.664,6.043,149.184
C03188=1157.086,-13.474,-46.567,179.661,6.042,149.185
C03189=1157.092,-13.724,-46.554,179.659,6.042,149.186
C03190=1157.097,-13.974,-46.541,179.656,6.041,149.186
C03191=1157.102,-14.224,-46.529,179.654,6.040,149.187
C03192=1157.107,-14.473,-46.517,179.651,6.040,149.187
C03193=1157.113,-14.723,-46.504,179.649,6.039,149.188
C03194=1157.118,-14.973,-46.490,179.646,6.039,149.189
C03195=1157.123,-15.222,-46.478,179.644,6.038,149.189
C03196=1157.128,-15.472,-46.465,179.642,6.037,149.190
C03197=1157.133,-15.721,-46.453,179.639,6.037,149.190
C03198=1157.139,-15.971,-46.441,179.637,6.036,149.191
C03199=1157.143,-16.221,-46.428,179.635,6.035,149.191
C03200=1157.148,-16.470,-46.415,179.632,6.035,149.192
C03201=1157.154,-16.720,-46.402,179.629,6.034,149.193
C03202=1157.159,-16.969,-46.389,179.627,6.034,149.193
C03203=1157.165,-17.219,-46.377,179.624,6.033,149.194
C03204=1157.169,-17.469,-46.364,179.622,6.032,149.194
C03205=1157.174,-17.718,-46.352,179.620,6.032,149.195
C03206=1157.179,-17.968,-46.339,179.617,6.031,149.196
C03207=1157.185,-18.218,-46.327,179.615,6.031,149.196
C03208=1157.190,-18.467,-46.315,179.613,6.030,149.197
C03209=1157.194,-18.717,-46.302,179.610,6.029,149.197
C03210=1157.200,-18.967,-46.289,179.608,6.029,149.198
C03211=1157.206,-19.216,-46.277,179.605,6.028,149.199
C03212=1157.211,-19.466,-46.264,179.603,6.027,149.199
C03213=1157.216,-19.715,-46.252,179.600,6.027,149.200
C03214=1157.221,-19.965,-46.240,179.598,6.026,149.200
C03215=1157.227,-20.214,-46.227,179.595,6.026,149.201
C03216=1157.231,-20.464,-46.214,179.593,6.025,149.201
C03217=1157.237,-20.714,-46.202,179.591,6.025,149.202
C03218=1157.242,-20.964,-46.190,179.588,6.024,149.203
C03219=1157.247,-21.213,-46.177,179.586,6.023,149.203
C03220=1157.252,-21.463,-46.165,179.583,6.022,149.204
C03221=1157.257,-21.712,-46.152,179.581,6.022,149.204
C03222=1157.262,-21.962,-46.140,179.579,6.021,149.205
C03223=1157.268,-22.211,-46.128,179.576,6.021,149.206
C03224=1157.272,-22.461,-46.115,179.574,6.020,149.206
C03225=1157.278,-22.711,-46.103,179.571,6.020,149.207
C03226=1157.283,-22.961,-46.091,179.569,6.019,149.207
C03227=1157.288,-23.210,-46.078,179.566,6.018,149.208
C03228=1157.294,-23.460,-46.066,179.564,6.018,149.208
C03229=1157.299,-23.709,-46.053,179.561,6.017,149.209
C03230=1157.305,-23.980,-46.040,179.559,6.017,149.210
C03231=1157.310,-24.249,-46.027,179.557,6.016,149.210
C03232=1157.316,-24.519,-46.014,179.554,6.015,149.211
C03233=1157.321,-24.790,-46.001,179.551,6.015,149.212
C03234=1157.326,-25.039,-45.988,179.549,6.014,149.212
C03235=1157.331,-25.288,-45.975,179.546,6.014,149.213
C03236=1157.337,-25.538,-45.964,179.544,6.013,149.213
C03237=1157.342,-25.788,-45.951,179.542,6.013,149.214
C03238=1157.347,-26.038,-45.939,179.539,6.012,149.215
C03239=1157.352,-26.287,-45.926,179.537,6.011,149.215
C03240=1157.358,-26.537,-45.915,179.535,6.011,149.216
C03241=1157.363,-26.787,-45.903,179.532,6.010,149.216
C03242=1157.368,-27.036,-45.890,179.530,6.009,149.217
C03243=1157.373,-27.286,-45.879,179.527,6.009,149.218
C03244=1157.378,-27.535,-45.866,179.525,6.008,149.218
C03245=1157.383,-27.785,-45.854,179.522,6.008,149.219
C03246=1157.389,-28.034,-45.842,179.520,6.007,149.219
C03247=1157.394,-28.284,-45.830,179.517,6.006,149.220
C03248=1157.399,-28.533,-45.817,179.515,6.006,149.221
C03249=1157.405,-28.783,-45.805,179.513,6.005,149.221
C03250=1157.409,-29.033,-45.794,179.510,6.005,149.222
C03251=1157.414,-29.282,-45.781,179.508,6.004,149.222
C03252=1157.420,-29.532,-45.770,179.505,6.004,149.223
C03253=1157.424,-29.782,-45.757,179.503,6.004,149.223
C03254=1157.430,-30.032,-45.745,179.501,6.003,149.224
C03255=1157.435,-30.282,-45.733,179.499,6.002,149.225
C03256=1157.440,-30.531,-45.721,179.496,6.002,149.225
C03257=1157.446,-30.780,-45.709,179.494,6.001,149.226
C03258=1157.451,-31.030,-45.697,179.491,6.001,149.226
C03259=1157.456,-31.280,-45.685,179.489,6.000,149.227
C03260=1157.462,-31.530,-45.673,179.486,5.999,149.228
C03261=1157.467,-31.780,-45.661,179.484,5.999,149.228
C03262=1157.471,-32.029,-45.649,179.481,5.998,149.229
C03263=1157.477,-32.279,-45.637,179.479,5.997,149.229
C03264=1157.482,-32.528,-45.625,179.477,5.997,149.230
C03265=1157.488,-32.778,-45.613,179.474,5.996,149.230
C03266=1157.492,-33.027,-45.601,179.472,5.996,149.231
C03267=1157.498,-33.277,-45.590,179.470,5.996,149.232
C03268=1157.503,-33.527,-45.578,179.467,5.995,149.232
C03269=1157.508,-33.777,-45.565,179.465,5.995,149.233
C03270=1157.513,-34.026,-45.554,179.463,5.994,149.233
C03271=1157.518,-34.276,-45.542,179.460,5.993,149.234
C03272=1157.524,-34.526,-45.530,179.458,5.993,149.235
C03273=1157.529,-34.776,-45.518,179.456,5.992,149.235
C03274=1157.533,-35.025,-45.506,179.453,5.992,149.236
C03275=1157.539,-35.275,-45.494,179.451,5.991,149.236
C03276=1157.544,-35.525,-45.482,179.448,5.991,149.237
C03277=1157.550,-35.774,-45.471,179.446,5.990,149.237
C03278=1157.555,-36.024,-45.459,179.443,5.989,149.238
C03279=1157.560,-36.273,-45.447,179.442,5.989,149.239
C03280=1157.566,-36.523,-45.435,179.439,5.989,149.239
C03281=1157.570,-36.773,-45.424,179.437,5.988,149.240
C03282=1157.576,-37.023,-45.412,179.434,5.988,149.241
C03283=1157.581,-37.273,-45.400,179.432,5.987,149.241
C03284=1157.586,-37.522,-45.389,179.429,5.986,149.242
C03285=1157.591,-37.771,-45.376,179.427,5.986,149.242
C03286=1157.597,-38.021,-45.365,179.424,5.985,149.243
C03287=1157.602,-38.270,-45.353,179.422,5.984,149.243
C03288=1157.607,-38.520,-45.341,179.420,5.984,149.244
C03289=1157.613,-38.770,-45.329,179.418,5.984,149.244
C03290=1157.617,-39.020,-45.318,179.415,5.984,149.245
C03291=1157.623,-39.270,-45.306,179.413,5.983,149.246
C03292=1157.627,-39.519,-45.295,179.410,5.982,149.246
C03293=1157.633,-39.769,-45.283,179.408,5.982,149.247
C03294=1157.639,-40.019,-45.272,179.406,5.981,149.248
C03295=1157.644,-40.268,-45.260,179.403,5.980,149.248
C03296=1157.649,-40.518,-45.248,179.401,5.980,149.249
C03297=1157.654,-40.768,-45.237,179.399,5.979,149.249
C03298=1157.659,-41.018,-45.225,179.397,5.980,149.250
C03299=1157.664,-41.268,-45.213,179.394,5.979,149.250
C03300=1157.669,-41.516,-45.202,179.392,5.978,149.251
C03301=1157.675,-41.766,-45.190,179.390,5.978,149.252
C03302=1157.680,-42.015,-45.179,179.387,5.977,149.252
C03303=1157.685,-42.265,-45.167,179.385,5.976,149.253
C03304=1157.691,-42.516,-45.156,179.382,5.976,149.253
C03305=1157.696,-42.765,-45.145,179.380,5.975,149.254
C03306=1157.701,-43.015,-45.133,179.378,5.976,149.255
C03307=1157.706,-43.264,-45.121,179.376,5.975,149.255
C03308=1157.712,-43.514,-45.110,179.373,5.974,149.256
C03309=1157.716,-43.764,-45.098,179.371,5.974,149.256
C03310=1157.722,-44.013,-45.087,179.368,5.973,149.257
C03311=1157.727,-44.263,-45.075,179.366,5.972,149.257
C03312=1157.732,-44.513,-45.064,179.363,5.972,149.258
C03313=1157.737,-44.762,-45.052,179.362,5.972,149.259
C03314=1157.743,-45.012,-45.040,179.359,5.972,149.259
C03315=1157.748,-45.261,-45.029,179.357,5.971,149.260
C03316=1157.753,-45.511,-45.018,179.354,5.970,149.260
C03317=1157.758,-45.761,-45.006,179.352,5.970,149.261
C03318=1157.764,-46.011,-44.995,179.350,5.969,149.261
C03319=1157.769,-46.260,-44.984,179.347,5.968,149.262
C03320=1157.774,-46.510,-44.972,179.345,5.968,149.263
C03321=1157.779,-46.760,-44.961,179.343,5.968,149.263
C03322=1157.785,-47.010,-44.949,179.341,5.967,149.264
C03323=1157.790,-47.259,-44.938,179.338,5.967,149.265
C03324=1157.795,-47.508,-44.927,179.336,5.966,149.265
C03325=1157.800,-47.759,-44.916,179.333,5.965,149.266
C03326=1157.805,-48.009,-44.904,179.331,5.965,149.266
C03327=1157.811,-48.258,-44.893,179.329,5.965,149.267
C03328=1157.816,-48.507,-44.882,179.327,5.964,149.267
C03329=1157.821,-48.757,-44.870,179.324,5.964,149.268
C03330=1157.827,-49.007,-44.860,179.322,5.963,149.269
C03331=1157.831,-49.257,-44.848,179.319,5.963,149.269
C03332=1157.837,-49.506,-44.836,179.317,5.962,149.270
C03333=1157.842,-49.756,-44.825,179.315,5.962,149.270
C03334=1157.848,-50.026,-44.813,179.313,5.961,149.271
C03335=1157.853,-50.297,-44.801,179.310,5.961,149.272
C03336=1157.859,-50.568,-44.789,179.307,5.961,149.272
C03337=1157.865,-50.839,-44.777,179.305,5.960,149.273
C03338=1157.870,-51.088,-44.765,179.302,5.959,149.273
C03339=1157.875,-51.338,-44.754,179.300,5.959,149.274
C03340=1157.881,-51.587,-44.743,179.298,5.958,149.275
C03341=1157.886,-51.837,-44.732,179.295,5.957,149.275
C03342=1157.890,-52.087,-44.721,179.293,5.958,149.276
C03343=1157.896,-52.336,-44.709,179.291,5.957,149.276
C03344=1157.901,-52.586,-44.699,179.289,5.957,149.277
C03345=1157.907,-52.836,-44.687,179.286,5.956,149.277
C03346=1157.912,-53.085,-44.676,179.284,5.956,149.278
C03347=1157.917,-53.336,-44.665,179.281,5.955,149.279
C03348=1157.922,-53.585,-44.654,179.279,5.955,149.279
C03349=1157.928,-53.834,-44.643,179.277,5.954,149.280
C03350=1157.933,-54.085,-44.632,179.275,5.954,149.281
C03351=1157.938,-54.334,-44.621,179.272,5.953,149.281
C03352=1157.944,-54.584,-44.610,179.270,5.953,149.282
C03353=1157.948,-54.834,-44.599,179.268,5.953,149.282
C03354=1157.954,-55.083,-44.588,179.265,5.952,149.283
C03355=1157.959,-55.333,-44.577,179.263,5.952,149.283
C03356=1157.964,-55.583,-44.565,179.261,5.951,149.284
C03357=1157.970,-55.832,-44.555,179.258,5.950,149.285
C03358=1157.975,-56.082,-44.544,179.257,5.950,149.285
C03359=1157.979,-56.332,-44.532,179.254,5.950,149.286
C03360=1157.986,-56.582,-44.522,179.252,5.949,149.286
C03361=1157.990,-56.831,-44.510,179.249,5.949,149.287
C03362=1157.996,-57.081,-44.500,179.247,5.948,149.287
C03363=1158.001,-57.330,-44.489,179.245,5.948,149.288
C03364=1158.006,-57.581,-44.478,179.243,5.948,149.289
C03365=1158.012,-57.830,-44.467,179.240,5.947,149.289
C03366=1158.017,-58.080,-44.456,179.238,5.946,149.290
C03367=1158.022,-58.329,-44.445,179.235,5.946,149.290
C03368=1158.027,-58.579,-44.435,179.234,5.946,149.291
C03369=1158.032,-58.829,-44.423,179.232,5.945,149.291
C03370=1158.038,-59.079,-44.413,179.229,5.945,149.292
C03371=1158.043,-59.328,-44.401,179.227,5.944,149.293
C03372=1158.048,-59.578,-44.391,179.224,5.944,149.293
C03373=1158.053,-59.827,-44.380,179.222,5.944,149.294
C03374=1158.059,-60.077,-44.369,179.220,5.943,149.295
C03375=1158.064,-60.327,-44.358,179.218,5.942,149.295
C03376=1158.069,-60.577,-44.347,179.215,5.942,149.296
C03377=1158.074,-60.826,-44.336,179.213,5.942,149.296
C03378=1158.079,-61.076,-44.326,179.211,5.942,149.297
C03379=1158.085,-61.326,-44.315,179.208,5.941,149.297
C03380=1158.089,-61.576,-44.304,179.206,5.940,149.298
C03381=1158.096,-61.825,-44.293,179.204,5.940,149.299
C03382=1158.100,-62.075,-44.282,179.202,5.940,149.299
C03383=1158.106,-62.325,-44.272,179.199,5.939,149.300
C03384=1158.111,-62.575,-44.261,179.197,5.939,149.300
C03385=1158.116,-62.824,-44.250,179.194,5.938,149.301
C03386=1158.121,-63.074,-44.240,179.193,5.938,149.301
C03387=1158.127,-63.323,-44.229,179.190,5.938,149.302
C03388=1158.132,-63.573,-44.218,179.188,5.937,149.303
C03389=1158.138,-63.823,-44.207,179.185,5.937,149.303
C03390=1158.143,-64.073,-44.196,179.183,5.936,149.304
C03391=1158.148,-64.322,-44.186,179.182,5.936,149.304
C03392=1158.153,-64.572,-44.175,179.179,5.935,149.305
C03393=1158.159,-64.821,-44.164,179.177,5.935,149.305
C03394=1158.164,-65.072,-44.154,179.174,5.934,149.306
C03395=1158.169,-65.321,-44.144,179.172,5.934,149.307
C03396=1158.174,-65.571,-44.133,179.170,5.934,149.307
C03397=1158.179,-65.820,-44.122,179.168,5.933,149.308
C03398=1158.184,-66.071,-44.112,179.165,5.933,149.309
C03399=1158.190,-66.320,-44.101,179.163,5.933,149.309
C03400=1158.195,-66.570,-44.090,179.161,5.932,149.309
C03401=1158.200,-66.819,-44.080,179.158,5.931,149.310
C03402=1158.205,-67.069,-44.069,179.156,5.931,149.311
C03403=1158.211,-67.319,-44.059,179.154,5.931,149.311
C03404=1158.216,-67.569,-44.048,179.152,5.930,149.312
C03405=1158.221,-67.818,-44.038,179.149,5.930,149.313
C03406=1158.226,-68.068,-44.027,179.147,5.929,149.313
C03407=1158.232,-68.318,-44.017,179.146,5.929,149.314
C03408=1158.237,-68.568,-44.007,179.143,5.929,149.314
C03409=1158.242,-68.817,-43.995,179.141,5.928,149.315
C03410=1158.248,-69.067,-43.985,179.138,5.928,149.315
C03411=1158.253,-69.317,-43.975,179.136,5.928,149.316
C03412=1158.258,-69.566,-43.964,179.134,5.927,149.317
C03413=1158.263,-69.817,-43.954,179.132,5.926,149.317
C03414=1158.269,-70.066,-43.943,179.130,5.927,149.318
C03415=1158.274,-70.315,-43.933,179.127,5.926,149.318
C03416=1158.279,-70.565,-43.922,179.125,5.925,149.319
C03417=1158.285,-70.815,-43.912,179.122,5.925,149.319
C03418=1158.290,-71.065,-43.901,179.121,5.925,149.320
C03419=1158.295,-71.315,-43.891,179.118,5.924,149.321
C03420=1158.301,-71.564,-43.881,179.116,5.924,149.321
C03421=1158.306,-71.814,-43.870,179.113,5.923,149.322
C03422=1158.311,-72.063,-43.859,179.112,5.923,149.322
C03423=1158.316,-72.314,-43.849,179.110,5.923,149.323
C03424=1158.322,-72.563,-43.839,179.107,5.922,149.324
C03425=1158.327,-72.813,-43.828,179.105,5.922,149.324
C03426=1158.332,-73.063,-43.818,179.103,5.922,149.325
C03427=1158.338,-73.313,-43.808,179.100,5.921,149.325
C03428=1158.344,-73.562,-43.797,179.098,5.920,149.326
C03429=1158.348,-73.812,-43.787,179.096,5.921,149.326
C03430=1158.354,-74.062,-43.777,179.094,5.920,149.327
C03431=1158.359,-74.311,-43.767,179.091,5.919,149.328
C03432=1158.364,-74.561,-43.756,179.090,5.919,149.328
C03433=1158.370,-74.811,-43.746,179.087,5.919,149.329
C03434=1158.375,-75.061,-43.736,179.085,5.918,149.329
C03435=1158.380,-75.311,-43.725,179.083,5.918,149.330
C03436=1158.386,-75.560,-43.715,179.081,5.918,149.330
C03437=1158.391,-75.810,-43.706,179.078,5.917,149.331
C03438=1158.397,-76.081,-43.694,179.076,5.917,149.332
C03439=1158.402,-76.352,-43.683,179.074,5.916,149.332
C03440=1158.408,-76.624,-43.672,179.071,5.916,149.333
C03441=1158.414,-76.895,-43.661,179.069,5.916,149.334
C03442=1158.419,-77.145,-43.650,179.067,5.915,149.334
C03443=1158.424,-77.394,-43.640,179.064,5.914,149.334
C03444=1158.430,-77.644,-43.630,179.062,5.914,149.335
C03445=1158.435,-77.894,-43.620,179.060,5.914,149.336
C03446=1158.440,-78.144,-43.609,179.057,5.914,149.336
C03447=1158.445,-78.393,-43.600,179.055,5.913,149.337
C03448=1158.451,-78.643,-43.589,179.054,5.913,149.337
C03449=1158.456,-78.893,-43.579,179.051,5.913,149.338
C03450=1158.461,-79.142,-43.569,179.049,5.912,149.339
C03451=1158.467,-79.392,-43.558,179.047,5.912,149.339
C03452=1158.472,-79.642,-43.549,179.045,5.911,149.340
C03453=1158.477,-79.892,-43.539,179.042,5.911,149.340
C03454=1158.483,-80.141,-43.529,179.040,5.911,149.341
C03455=1158.488,-80.391,-43.518,179.038,5.910,149.341
C03456=1158.493,-80.641,-43.509,179.035,5.910,149.342
C03457=1158.498,-80.891,-43.498,179.033,5.909,149.343
C03458=1158.504,-81.140,-43.488,179.032,5.909,149.343
C03459=1158.509,-81.390,-43.478,179.029,5.909,149.344
C03460=1158.514,-81.640,-43.469,179.027,5.908,149.344
C03461=1158.520,-81.890,-43.458,179.025,5.908,149.345
C03462=1158.525,-82.139,-43.448,179.022,5.908,149.345
C03463=1158.531,-82.389,-43.438,179.020,5.907,149.346
C03464=1158.535,-82.639,-43.428,179.018,5.907,149.347
C03465=1158.541,-82.889,-43.419,179.016,5.906,149.347
C03466=1158.547,-83.138,-43.408,179.013,5.906,149.348
C03467=1158.551,-83.388,-43.399,179.012,5.906,149.348
C03468=1158.556,-83.638,-43.388,179.010,5.905,149.349
C03469=1158.562,-83.887,-43.378,179.007,5.905,149.350
C03470=1158.567,-84.137,-43.369,179.005,5.905,149.350
C03471=1158.573,-84.387,-43.359,179.003,5.905,149.351
C03472=1158.578,-84.637,-43.348,179.000,5.904,149.351
C03473=1158.583,-84.886,-43.339,178.999,5.904,149.352
C03474=1158.589,-85.136,-43.329,178.996,5.903,149.352
C03475=1158.594,-85.386,-43.319,178.994,5.903,149.353
C03476=1158.599,-85.635,-43.309,178.992,5.903,149.353
C03477=1158.604,-85.885,-43.299,178.990,5.902,149.354
C03478=1158.610,-86.136,-43.289,178.988,5.902,149.355
C03479=1158.615,-86.385,-43.280,178.985,5.902,149.355
C03480=1158.620,-86.634,-43.269,178.983,5.901,149.356
C03481=1158.626,-86.885,-43.260,178.981,5.900,149.356
C03482=1158.631,-87.135,-43.250,178.979,5.901,149.357
C03483=1158.636,-87.384,-43.240,178.977,5.900,149.357
C03484=1158.641,-87.634,-43.231,178.975,5.899,149.358
C03485=1158.647,-87.883,-43.221,178.973,5.900,149.359
C03486=1158.653,-88.133,-43.210,178.970,5.899,149.359
C03487=1158.658,-88.383,-43.202,178.968,5.899,149.360
C03488=1158.663,-88.633,-43.191,178.966,5.899,149.360
C03489=1158.668,-88.882,-43.181,178.964,5.898,149.361
C03490=1158.673,-89.133,-43.172,178.962,5.898,149.361
C03491=1158.679,-89.382,-43.162,178.960,5.897,149.362
C03492=1158.684,-89.631,-43.152,178.957,5.897,149.362
C03493=1158.690,-89.881,-43.143,178.955,5.897,149.363
C03494=1158.694,-90.131,-43.133,178.953,5.896,149.364
C03495=1158.700,-90.382,-43.123,178.951,5.896,149.364
C03496=1158.705,-90.631,-43.113,178.949,5.896,149.365
C03497=1158.710,-90.880,-43.103,178.947,5.895,149.365
C03498=1158.716,-91.130,-43.094,178.944,5.895,149.366
C03499=1158.721,-91.380,-43.084,178.942,5.895,149.367
C03500=1158.727,-91.630,-43.075,178.940,5.894,149.367
C03501=1158.731,-91.880,-43.065,178.938,5.894,149.368
C03502=1158.737,-92.130,-43.055,178.936,5.894,149.368
C03503=1158.742,-92.379,-43.046,178.934,5.893,149.369
C03504=1158.748,-92.629,-43.035,178.932,5.893,149.369
C03505=1158.753,-92.879,-43.026,178.929,5.893,149.370
C03506=1158.758,-93.128,-43.016,178.927,5.892,149.370
C03507=1158.764,-93.378,-43.007,178.925,5.892,149.371
C03508=1158.769,-93.628,-42.997,178.923,5.891,149.372
C03509=1158.774,-93.877,-42.988,178.921,5.891,149.372
C03510=1158.780,-94.127,-42.978,178.919,5.891,149.373
C03511=1158.785,-94.377,-42.969,178.917,5.890,149.373
C03512=1158.790,-94.627,-42.959,178.915,5.890,149.374
C03513=1158.795,-94.877,-42.950,178.912,5.890,149.374
C03514=1158.801,-95.126,-42.939,178.910,5.889,149.375
C03515=1158.806,-95.376,-42.931,178.908,5.889,149.375
C03516=1158.812,-95.626,-42.921,178.906,5.889,149.376
C03517=1158.817,-95.876,-42.911,178.904,5.889,149.377
C03518=1158.822,-96.126,-42.903,178.902,5.888,149.377
C03519=1158.828,-96.375,-42.892,178.899,5.888,149.378
C03520=1158.833,-96.625,-42.883,178.898,5.888,149.378
C03521=1158.838,-96.874,-42.873,178.896,5.887,149.379
C03522=1158.844,-97.124,-42.864,178.893,5.887,149.379
C03523=1158.849,-97.374,-42.854,178.891,5.887,149.380
C03524=1158.854,-97.624,-42.845,178.889,5.886,149.380
C03525=1158.860,-97.874,-42.836,178.887,5.886,149.381
C03526=1158.865,-98.123,-42.826,178.885,5.886,149.382
C03527=1158.870,-98.373,-42.817,178.883,5.885,149.382
C03528=1158.876,-98.623,-42.808,178.881,5.885,149.383
C03529=1158.880,-98.873,-42.798,178.878,5.884,149.383
C03530=1158.886,-99.123,-42.788,178.877,5.884,149.384
C03531=1158.891,-99.372,-42.779,178.874,5.884,149.385
C03532=1158.896,-99.622,-42.770,178.872,5.883,149.385
C03533=1158.902,-99.872,-42.760,178.870,5.883,149.385
C03534=1158.907,-100.122,-42.751,178.868,5.883,149.386
C03535=1158.912,-100.372,-42.742,178.866,5.883,149.387
C03536=1158.918,-100.622,-42.732,178.864,5.882,149.387
C03537=1158.923,-100.871,-42.723,178.861,5.882,149.388
C03538=1158.929,-101.121,-42.713,178.860,5.882,149.388
C03539=1158.934,-101.371,-42.704,178.857,5.881,149.389
C03540=1158.939,-101.621,-42.695,178.855,5.881,149.390
C03541=1158.945,-101.870,-42.685,178.853,5.881,149.390
C03542=1158.951,-102.142,-42.675,178.851,5.880,149.391
C03543=1158.957,-102.414,-42.666,178.849,5.880,149.391
C03544=1158.962,-102.686,-42.656,178.847,5.880,149.392
C03545=1158.968,-102.958,-42.645,178.844,5.879,149.392
C03546=1158.974,-103.208,-42.636,178.842,5.879,149.393
C03547=1158.979,-103.458,-42.627,178.840,5.879,149.394
C03548=1158.984,-103.707,-42.617,178.837,5.878,149.394
C03549=1158.989,-103.957,-42.608,178.836,5.878,149.395
C03550=1158.995,-104.207,-42.599,178.833,5.878,149.395
C03551=1159.000,-104.457,-42.590,178.832,5.878,149.396
C03552=1159.005,-104.706,-42.580,178.829,5.877,149.396
C03553=1159.011,-104.956,-42.571,178.827,5.876,149.397
C03554=1159.016,-105.206,-42.562,178.825,5.877,149.397
C03555=1159.021,-105.456,-42.553,178.823,5.876,149.398
C03556=1159.027,-105.705,-42.545,178.821,5.876,149.398
C03557=1159.032,-105.955,-42.534,178.819,5.876,149.399
C03558=1159.038,-106.205,-42.525,178.817,5.876,149.400
C03559=1159.043,-106.455,-42.517,178.815,5.875,149.400
C03560=1159.048,-106.704,-42.508,178.813,5.874,149.401
C03561=1159.054,-106.955,-42.498,178.811,5.875,149.401
C03562=1159.059,-107.204,-42.489,178.808,5.874,149.402
C03563=1159.064,-107.454,-42.480,178.807,5.874,149.402
C03564=1159.069,-107.703,-42.471,178.804,5.873,149.403
C03565=1159.074,-107.953,-42.462,178.803,5.873,149.404
C03566=1159.080,-108.204,-42.452,178.800,5.873,149.404
C03567=1159.085,-108.453,-42.443,178.798,5.872,149.404
C03568=1159.090,-108.703,-42.435,178.796,5.872,149.405
C03569=1159.096,-108.952,-42.426,178.794,5.872,149.406
C03570=1159.102,-109.203,-42.417,178.792,5.872,149.406
C03571=1159.107,-109.452,-42.408,178.790,5.871,149.407
C03572=1159.112,-109.702,-42.398,178.788,5.871,149.407
C03573=1159.117,-109.951,-42.389,178.786,5.871,149.408
C03574=1159.122,-110.201,-42.380,178.784,5.871,149.408
C03575=1159.128,-110.451,-42.371,178.782,5.870,149.409
C03576=1159.133,-110.701,-42.362,178.779,5.869,149.410
C03577=1159.139,-110.950,-42.353,178.778,5.869,149.410
C03578=1159.144,-111.200,-42.344,178.775,5.869,149.411
C03579=1159.150,-111.450,-42.336,178.773,5.869,149.411
C03580=1159.155,-111.700,-42.327,178.771,5.868,149.412
C03581=1159.160,-111.950,-42.318,178.770,5.868,149.412
C03582=1159.166,-112.200,-42.308,178.767,5.868,149.413
C03583=1159.171,-112.450,-42.299,178.765,5.868,149.413
C03584=1159.176,-112.700,-42.290,178.763,5.867,149.414
C03585=1159.182,-112.949,-42.282,178.761,5.867,149.414
C03586=1159.187,-113.199,-42.273,178.759,5.867,149.415
C03587=1159.192,-113.449,-42.264,178.757,5.866,149.416
C03588=1159.197,-113.698,-42.255,178.755,5.866,149.416
C03589=1159.203,-113.948,-42.246,178.753,5.865,149.417
C03590=1159.209,-114.198,-42.237,178.751,5.866,149.417
C03591=1159.214,-114.448,-42.228,178.749,5.865,149.418
C03592=1159.219,-114.697,-42.219,178.747,5.865,149.418
C03593=1159.225,-114.947,-42.211,178.745,5.864,149.419
C03594=1159.230,-115.197,-42.202,178.743,5.865,149.419
C03595=1159.235,-115.447,-42.193,178.741,5.864,149.420
C03596=1159.241,-115.696,-42.184,178.738,5.863,149.420
C03597=1159.246,-115.946,-42.175,178.737,5.863,149.421
C03598=1159.251,-116.196,-42.166,178.734,5.863,149.422
C03599=1159.257,-116.446,-42.158,178.733,5.863,149.422
C03600=1159.262,-116.696,-42.149,178.730,5.862,149.423
C03601=1159.268,-116.946,-42.140,178.729,5.862,149.423
C03602=1159.273,-117.196,-42.131,178.726,5.862,149.424
C03603=1159.279,-117.445,-42.122,178.724,5.862,149.424
C03604=1159.284,-117.695,-42.113,178.722,5.861,149.425
C03605=1159.289,-117.945,-42.105,178.721,5.861,149.425
C03606=1159.295,-118.194,-42.096,178.718,5.861,149.426
C03607=1159.300,-118.444,-42.087,178.716,5.861,149.426
C03608=1159.305,-118.695,-42.079,178.714,5.860,149.427
C03609=1159.310,-118.944,-42.070,178.713,5.860,149.427
C03610=1159.316,-119.194,-42.062,178.710,5.859,149.428
C03611=1159.321,-119.443,-42.053,178.708,5.860,149.429
C03612=1159.327,-119.693,-42.044,178.706,5.859,149.429
C03613=1159.332,-119.943,-42.035,178.704,5.858,149.430
C03614=1159.337,-120.194,-42.027,178.702,5.858,149.430
C03615=1159.343,-120.443,-42.018,178.700,5.858,149.431
C03616=1159.348,-120.693,-42.009,178.698,5.858,149.431
C03617=1159.353,-120.942,-42.000,178.696,5.857,149.432
C03618=1159.358,-121.192,-41.991,178.694,5.857,149.432
C03619=1159.364,-121.442,-41.984,178.692,5.857,149.433
C03620=1159.370,-121.692,-41.975,178.690,5.857,149.433
C03621=1159.375,-121.942,-41.966,178.688,5.856,149.434
C03622=1159.381,-122.191,-41.957,178.686,5.856,149.434
C03623=1159.386,-122.441,-41.948,178.684,5.856,149.435
C03624=1159.390,-122.691,-41.941,178.682,5.856,149.436
C03625=1159.396,-122.941,-41.932,178.680,5.855,149.436
C03626=1159.401,-123.190,-41.923,178.678,5.855,149.437
C03627=1159.407,-123.440,-41.914,178.676,5.855,149.437
C03628=1159.412,-123.690,-41.906,178.674,5.855,149.438
C03629=1159.417,-123.940,-41.897,178.672,5.854,149.438
C03630=1159.423,-124.189,-41.889,178.670,5.854,149.439
C03631=1159.428,-124.440,-41.881,178.668,5.853,149.439
C03632=1159.434,-124.690,-41.872,178.666,5.853,149.440
C03633=1159.439,-124.939,-41.863,178.664,5.853,149.440
C03634=1159.445,-125.189,-41.854,178.662,5.853,149.441
C03635=1159.450,-125.439,-41.846,178.660,5.852,149.441
C03636=1159.455,-125.688,-41.838,178.658,5.852,149.442
C03637=1159.460,-125.938,-41.829,178.656,5.852,149.442
C03638=1159.466,-126.188,-41.821,178.654,5.852,149.443
C03639=1159.471,-126.437,-41.813,178.652,5.851,149.443
C03640=1159.477,-126.687,-41.804,178.650,5.851,149.444
C03641=1159.482,-126.938,-41.796,178.648,5.851,149.445
C03642=1159.488,-127.187,-41.787,178.646,5.851,149.445
C03643=1159.493,-127.437,-41.779,178.644,5.850,149.446
C03644=1159.499,-127.687,-41.770,178.643,5.850,149.446
C03645=1159.504,-127.936,-41.762,178.640,5.850,149.447
C03646=1159.083,-127.948,-41.804,178.637,5.853,149.448
C03647=1159.077,-127.698,-41.812,178.639,5.853,149.448
